# B&R Automation Studio project OpcUaSample410_BrbLibUa103 (part 5)

#### BrbDtStructCompare.c - Vergleicht zwei DtStructures
```c
/********************************************************************
 * COPYRIGHT -- Bernecker + Rainer
 ********************************************************************
 * Library: BrbLib
 * File: BrbDtStructCompare.c
 * Author: niedermeierr
 * Created: December 11, 2013
 ********************************************************************
 * Implementation of library BrbLib
 ********************************************************************/

#include <bur/plctypes.h>
#ifdef __cplusplus
	extern "C"
	{
#endif

	#include "BrbLib.h"

#ifdef __cplusplus
	};
#endif

// NOLINTBEGIN(readability-*, bugprone-easily-swappable-parameters, clang-diagnostic-invalid-utf8, clang-diagnostic-invalid-source-encoding, clang-diagnostic-pointer-arith, clang-diagnostic-strict-prototypes, hicpp-uppercase-literal-suffix, cppcoreguidelines-*, performance-*)

/* Vergleicht zwei DtStructures */
plcbit BrbDtStructCompare(struct DTStructure* pDtStruct1, enum BrbTimeAndDateCompare_ENUM eCompare, struct DTStructure* pDtStruct2) // NOLINT(readability-function-cognitive-complexity)
{
	// Prüfung der Parameter
	if(pDtStruct1 == 0)
	{
		return 0;
	}
	if(pDtStruct2 == 0)
	{
		return 0;
	}
	// Vergleich
	BOOL bResult = 0;
	switch(eCompare) // NOLINT(hicpp-multiway-paths-covered)
	{
		case eBRB_TAD_COMPARE_YOUNGER:
			if(pDtStruct1->year < pDtStruct2->year)
			{
				bResult = 1;
			}
			else if(pDtStruct1->year == pDtStruct2->year)
			{
				if(pDtStruct1->month < pDtStruct2->month)
				{
					bResult = 1;
				}
				else if(pDtStruct1->month == pDtStruct2->month)
				{
					if(pDtStruct1->day < pDtStruct2->day)
					{
						bResult = 1;
					}
					else if(pDtStruct1->day == pDtStruct2->day)
					{
						if(pDtStruct1->hour < pDtStruct2->hour)
						{
							bResult = 1;
						}
						else if(pDtStruct1->hour == pDtStruct2->hour)
						{
							if(pDtStruct1->minute < pDtStruct2->minute)
							{
								bResult = 1;
							}
							else if(pDtStruct1->minute == pDtStruct2->minute)
							{
								if(pDtStruct1->second < pDtStruct2->second)
								{
									bResult = 1;
								}
								else if(pDtStruct1->second == pDtStruct2->second)
								{
									if(pDtStruct1->millisec < pDtStruct2->millisec)
									{
										bResult = 1;
									}
									else if(pDtStruct1->millisec == pDtStruct2->millisec)
									{
										if(pDtStruct1->microsec < pDtStruct2->microsec)
										{
											bResult = 1;
										}
										else if(pDtStruct1->microsec == pDtStruct2->microsec)
										{
											bResult = 0;
										}
									}
								}
							}
						}
					}
				}
			}
			break;

		case eBRB_TAD_COMPARE_YOUNGEREQUAL:
			// NOLINTBEGIN(bugprone-branch-clone)
			if(pDtStruct1->year < pDtStruct2->year)
			{
				bResult = 1;
			}
			else if(pDtStruct1->year == pDtStruct2->year)
			{
				if(pDtStruct1->month < pDtStruct2->month)
				{
					bResult = 1;
				}
				else if(pDtStruct1->month == pDtStruct2->month)
				{
					if(pDtStruct1->day < pDtStruct2->day)
					{
						bResult = 1;
					}
					else if(pDtStruct1->day == pDtStruct2->day)
					{
						if(pDtStruct1->hour < pDtStruct2->hour)
						{
							bResult = 1;
						}
						else if(pDtStruct1->hour == pDtStruct2->hour)
						{
							if(pDtStruct1->minute < pDtStruct2->minute)
							{
								bResult = 1;
							}
							else if(pDtStruct1->minute == pDtStruct2->minute)
							{
								if(pDtStruct1->second < pDtStruct2->second)
								{
									bResult = 1;
								}
								else if(pDtStruct1->second == pDtStruct2->second)
								{
									if(pDtStruct1->millisec < pDtStruct2->millisec)
									{
										bResult = 1;
									}
									else if(pDtStruct1->millisec == pDtStruct2->millisec)
									{
										if(pDtStruct1->microsec < pDtStruct2->microsec)
										{
											bResult = 1;
										}
										else if(pDtStruct1->microsec == pDtStruct2->microsec)
										{
											bResult = 1;
										}
									}
								}
							}
						}
					}
				}
			}
			// NOLINTEND(bugprone-branch-clone)
			break;

		case eBRB_TAD_COMPARE_EQUAL:
			if((pDtStruct1->year == pDtStruct2->year) &&
				(pDtStruct1->month == pDtStruct2->month) &&
				(pDtStruct1->day == pDtStruct2->day) &&
				(pDtStruct1->hour == pDtStruct2->hour) &&
				(pDtStruct1->minute == pDtStruct2->minute) &&
				(pDtStruct1->second == pDtStruct2->second) &&
				(pDtStruct1->millisec == pDtStruct2->millisec) &&
				(pDtStruct1->microsec == pDtStruct2->microsec)
				)
			{
				bResult = 1;
			}
			break;

		case eBRB_TAD_COMPARE_OLDEREQUAL:
			// NOLINTBEGIN(bugprone-branch-clone)
			if(pDtStruct1->year > pDtStruct2->year)
			{
				bResult = 1;
			}
			else if(pDtStruct1->year == pDtStruct2->year)
			{
				if(pDtStruct1->month > pDtStruct2->month)
				{
					bResult = 1;
				}
				else if(pDtStruct1->month == pDtStruct2->month)
				{
					if(pDtStruct1->day > pDtStruct2->day)
					{
						bResult = 1;
					}
					else if(pDtStruct1->day == pDtStruct2->day)
					{
						if(pDtStruct1->hour > pDtStruct2->hour)
						{
							bResult = 1;
						}
						else if(pDtStruct1->hour == pDtStruct2->hour)
						{
							if(pDtStruct1->minute > pDtStruct2->minute)
							{
								bResult = 1;
							}
							else if(pDtStruct1->minute == pDtStruct2->minute)
							{
								if(pDtStruct1->second > pDtStruct2->second)
								{
									bResult = 1;
								}
								else if(pDtStruct1->second == pDtStruct2->second)
								{
									if(pDtStruct1->millisec > pDtStruct2->millisec)
									{
										bResult = 1;
									}
									else if(pDtStruct1->millisec == pDtStruct2->millisec)
									{
										if(pDtStruct1->microsec > pDtStruct2->microsec)
										{
											bResult = 1;
										}
										else if(pDtStruct1->microsec == pDtStruct2->microsec)
										{
											bResult = 1;
										}
									}
								}
							}
						}
					}
				}
			}
			// NOLINTEND(bugprone-branch-clone)
			break;

		case eBRB_TAD_COMPARE_OLDER:
			if(pDtStruct1->year > pDtStruct2->year)
			{
				bResult = 1;
			}
			else if(pDtStruct1->year == pDtStruct2->year)
			{
				if(pDtStruct1->month > pDtStruct2->month)
				{
					bResult = 1;
				}
				else if(pDtStruct1->month == pDtStruct2->month)
				{
					if(pDtStruct1->day > pDtStruct2->day)
					{
						bResult = 1;
					}
					else if(pDtStruct1->day == pDtStruct2->day)
					{
						if(pDtStruct1->hour > pDtStruct2->hour)
						{
							bResult = 1;
						}
						else if(pDtStruct1->hour == pDtStruct2->hour)
						{
							if(pDtStruct1->minute > pDtStruct2->minute)
							{
								bResult = 1;
							}
							else if(pDtStruct1->minute == pDtStruct2->minute)
							{
								if(pDtStruct1->second > pDtStruct2->second)
								{
									bResult = 1;
								}
								else if(pDtStruct1->second == pDtStruct2->second)
								{
									if(pDtStruct1->millisec > pDtStruct2->millisec)
									{
										bResult = 1;
									}
									else if(pDtStruct1->millisec == pDtStruct2->millisec)
									{
										if(pDtStruct1->microsec > pDtStruct2->microsec)
										{
											bResult = 1;
										}
										else if(pDtStruct1->microsec == pDtStruct2->microsec)
										{
											bResult = 0;
										}
									}
								}
							}
						}
					}
				}
			}
			break;

	}

	return bResult;
}

// NOLINTEND(readability-*, bugprone-easily-swappable-parameters, clang-diagnostic-invalid-utf8, clang-diagnostic-invalid-source-encoding, clang-diagnostic-pointer-arith, clang-diagnostic-strict-prototypes, hicpp-uppercase-literal-suffix, cppcoreguidelines-*, performance-*)
```

#### BrbDtStructAddDays.c - Addiert zu einer DTStructure die angegebenen Sekunden
```c
/********************************************************************
 * COPYRIGHT -- Bernecker + Rainer
 ********************************************************************
 * Library: BrbLib
 * File: BrbDtStructAddSeconds.c
 * Author: niedermeierr
 * Created: September 08, 2021
 ********************************************************************
 * Implementation of library BrbLib
 ********************************************************************/

#include <bur/plctypes.h>
#ifdef __cplusplus
	extern "C"
	{
#endif

#include "BrbLib.h"
#include <AnsiCFunc.h>

#ifdef __cplusplus
	};
#endif

// NOLINTBEGIN(readability-*, bugprone-easily-swappable-parameters, clang-diagnostic-invalid-utf8, clang-diagnostic-invalid-source-encoding, clang-diagnostic-pointer-arith, clang-diagnostic-strict-prototypes, hicpp-uppercase-literal-suffix, cppcoreguidelines-*, performance-*)

/* Addiert zu einer DTStructure die angegebenen Sekunden */
plcdt BrbDtStructAddDays(struct DTStructure* pDtStruct, signed long nDays)
{
	// Prüfung der Parameter
	if(pDtStruct == 0)
	{
		return 0;
	}
	// Addieren
	UINT nMilliSecondsBefore = pDtStruct->millisec;
	UINT nMicroSecondsBefore = pDtStruct->microsec;
	DATE_AND_TIME dtTime = DTStructure_TO_DT((UDINT)pDtStruct);
	// Es müssen Sekunden addiert werden. Durch eine Multiplikation der Stunden mit 60s*60m*24h = 86400s könnte der Bereich eines Dint nicht mehr ausreichen
	// Daher wird eine Schleife durchlaufen.
	UDINT nLoop = 0;
	if(nDays < 0)
	{
		for(nLoop=0; nLoop<(UDINT)abs(nDays); nLoop++)
		{
			dtTime = dtTime - nBRB_SECONDS_PER_DAY;
		}
	}
	else
	{
		for(nLoop=0; nLoop<(UDINT)abs(nDays); nLoop++)
		{
			dtTime = dtTime + nBRB_SECONDS_PER_DAY;
		}
	}
	DT_TO_DTStructure(dtTime, (UDINT)pDtStruct);
	pDtStruct->millisec = nMilliSecondsBefore;
	pDtStruct->microsec = nMicroSecondsBefore;
	return dtTime;
}

// NOLINTEND(readability-*, bugprone-easily-swappable-parameters, clang-diagnostic-invalid-utf8, clang-diagnostic-invalid-source-encoding, clang-diagnostic-pointer-arith, clang-diagnostic-strict-prototypes, hicpp-uppercase-literal-suffix, cppcoreguidelines-*, performance-*)
```

#### BrbDtStructAddHours.c - Addiert zu einer DTStructure die angegebenen Sekunden
```c
/********************************************************************
 * COPYRIGHT -- Bernecker + Rainer
 ********************************************************************
 * Library: BrbLib
 * File: BrbDtStructAddSeconds.c
 * Author: niedermeierr
 * Created: September 08, 2021
 ********************************************************************
 * Implementation of library BrbLib
 ********************************************************************/

#include <bur/plctypes.h>
#ifdef __cplusplus
	extern "C"
	{
#endif

#include "BrbLib.h"
#include <AnsiCFunc.h>

#ifdef __cplusplus
	};
#endif

// NOLINTBEGIN(readability-*, bugprone-easily-swappable-parameters, clang-diagnostic-invalid-utf8, clang-diagnostic-invalid-source-encoding, clang-diagnostic-pointer-arith, clang-diagnostic-strict-prototypes, hicpp-uppercase-literal-suffix, cppcoreguidelines-*, performance-*)

/* Addiert zu einer DTStructure die angegebenen Sekunden */
plcdt BrbDtStructAddHours(struct DTStructure* pDtStruct, signed long nHours)
{
	// Prüfung der Parameter
	if(pDtStruct == 0)
	{
		return 0;
	}
	// Addieren
	UINT nMilliSecondsBefore = pDtStruct->millisec;
	UINT nMicroSecondsBefore = pDtStruct->microsec;
	DATE_AND_TIME dtTime = DTStructure_TO_DT((UDINT)pDtStruct);
	// Es müssen Sekunden addiert werden. Durch eine Multiplikation der Stunden mit 60s*60m = 3600s könnte der Bereich eines Dint nicht mehr ausreichen
	// Daher wird eine Schleife durchlaufen.
	UDINT nLoop = 0;
	if(nHours < 0)
	{
		for(nLoop=0; nLoop<(UDINT)abs(nHours); nLoop++)
		{
			dtTime = dtTime - nBRB_SECONDS_PER_HOUR;
		}
	}
	else
	{
		for(nLoop=0; nLoop<(UDINT)abs(nHours); nLoop++)
		{
			dtTime = dtTime + nBRB_SECONDS_PER_HOUR;
		}
	}
	DT_TO_DTStructure(dtTime, (UDINT)pDtStruct);
	pDtStruct->millisec = nMilliSecondsBefore;
	pDtStruct->microsec = nMicroSecondsBefore;
	return dtTime;
}

// NOLINTEND(readability-*, bugprone-easily-swappable-parameters, clang-diagnostic-invalid-utf8, clang-diagnostic-invalid-source-encoding, clang-diagnostic-pointer-arith, clang-diagnostic-strict-prototypes, hicpp-uppercase-literal-suffix, cppcoreguidelines-*, performance-*)
```

#### BrbDtStructAddMinutes.c - Addiert zu einer DTStructure die angegebenen Sekunden
```c
/********************************************************************
 * COPYRIGHT -- Bernecker + Rainer
 ********************************************************************
 * Library: BrbLib
 * File: BrbDtStructAddSeconds.c
 * Author: niedermeierr
 * Created: September 08, 2021
 ********************************************************************
 * Implementation of library BrbLib
 ********************************************************************/

#include <bur/plctypes.h>
#ifdef __cplusplus
	extern "C"
	{
#endif

#include "BrbLib.h"
#include <AnsiCFunc.h>

#ifdef __cplusplus
	};
#endif

// NOLINTBEGIN(readability-*, bugprone-easily-swappable-parameters, clang-diagnostic-invalid-utf8, clang-diagnostic-invalid-source-encoding, clang-diagnostic-pointer-arith, clang-diagnostic-strict-prototypes, hicpp-uppercase-literal-suffix, cppcoreguidelines-*, performance-*)

/* Addiert zu einer DTStructure die angegebenen Sekunden */
plcdt BrbDtStructAddMinutes(struct DTStructure* pDtStruct, signed long nMinutes)
{
	// Prüfung der Parameter
	if(pDtStruct == 0)
	{
		return 0;
	}
	// Addieren
	UINT nMilliSecondsBefore = pDtStruct->millisec;
	UINT nMicroSecondsBefore = pDtStruct->microsec;
	DATE_AND_TIME dtTime = DTStructure_TO_DT((UDINT)pDtStruct);
	// Es müssen Sekunden addiert werden. Durch eine Multiplikation der Minuten mit 60s könnte der Bereich eines Dint nicht mehr ausreichen
	// Daher wird eine Schleife durchlaufen.
	UDINT nLoop = 0;
	if(nMinutes < 0)
	{
		for(nLoop=0; nLoop<(UDINT)abs(nMinutes); nLoop++)
		{
			dtTime = dtTime - nBRB_SECONDS_PER_MINUTE;
		}
	}
	else
	{
		for(nLoop=0; nLoop<(UDINT)abs(nMinutes); nLoop++)
		{
			dtTime = dtTime + nBRB_SECONDS_PER_MINUTE;
		}
	}
	DT_TO_DTStructure(dtTime, (UDINT)pDtStruct);
	pDtStruct->millisec = nMilliSecondsBefore;
	pDtStruct->microsec = nMicroSecondsBefore;
	return dtTime;
}

// NOLINTEND(readability-*, bugprone-easily-swappable-parameters, clang-diagnostic-invalid-utf8, clang-diagnostic-invalid-source-encoding, clang-diagnostic-pointer-arith, clang-diagnostic-strict-prototypes, hicpp-uppercase-literal-suffix, cppcoreguidelines-*, performance-*)
```

#### BrbDtStructAddSeconds.c - Addiert zu einer DTStructure die angegebenen Sekunden
```c
/********************************************************************
 * COPYRIGHT -- Bernecker + Rainer
 ********************************************************************
 * Library: BrbLib
 * File: BrbDtStructAddSeconds.c
 * Author: niedermeierr
 * Created: September 08, 2021
 ********************************************************************
 * Implementation of library BrbLib
 ********************************************************************/

#include <bur/plctypes.h>
#ifdef __cplusplus
	extern "C"
	{
#endif

	#include "BrbLib.h"

#ifdef __cplusplus
	};
#endif

// NOLINTBEGIN(readability-*, bugprone-easily-swappable-parameters, clang-diagnostic-invalid-utf8, clang-diagnostic-invalid-source-encoding, clang-diagnostic-pointer-arith, clang-diagnostic-strict-prototypes, hicpp-uppercase-literal-suffix, cppcoreguidelines-*, performance-*)

/* Addiert zu einer DTStructure die angegebenen Sekunden */
plcdt BrbDtStructAddSeconds(struct DTStructure* pDtStruct, signed long nSeconds)
{
	// Prüfung der Parameter
	if(pDtStruct == 0)
	{
		return 0;
	}
	// Addieren
	UINT nMilliSecondsBefore = pDtStruct->millisec;
	UINT nMicroSecondsBefore = pDtStruct->microsec;
	DATE_AND_TIME dtTime = DTStructure_TO_DT((UDINT)pDtStruct);
	if(nSeconds < 0)
	{
		dtTime = dtTime - (UDINT)(nSeconds * -1);
	}
	else
	{
		dtTime = dtTime + (UDINT)nSeconds;
	}
	DT_TO_DTStructure(dtTime, (UDINT)pDtStruct);
	pDtStruct->millisec = nMilliSecondsBefore;
	pDtStruct->microsec = nMicroSecondsBefore;
	return dtTime;
}

// NOLINTEND(readability-*, bugprone-easily-swappable-parameters, clang-diagnostic-invalid-utf8, clang-diagnostic-invalid-source-encoding, clang-diagnostic-pointer-arith, clang-diagnostic-strict-prototypes, hicpp-uppercase-literal-suffix, cppcoreguidelines-*, performance-*)
```

#### BrbDtStructAddMilliseconds.c - Addiert zu einer DTStructure die angegebenen Millisekunden
```c
/********************************************************************
 * COPYRIGHT -- Bernecker + Rainer
 ********************************************************************
 * Library: BrbLib
 * File: BrbDtStructAddMilliseconds.c
 * Author: niedermeierr
 * Created: December 11, 2013
 ********************************************************************
 * Implementation of library BrbLib
 ********************************************************************/

#include <bur/plctypes.h>
#ifdef __cplusplus
	extern "C"
	{
#endif

	#include "BrbLib.h"

#ifdef __cplusplus
	};
#endif

// NOLINTBEGIN(readability-*, bugprone-easily-swappable-parameters, clang-diagnostic-invalid-utf8, clang-diagnostic-invalid-source-encoding, clang-diagnostic-pointer-arith, clang-diagnostic-strict-prototypes, hicpp-uppercase-literal-suffix, cppcoreguidelines-*, performance-*)

/* Addiert zu einer DTStructure die angegebenen Millisekunden */
plcdt BrbDtStructAddMilliseconds(struct DTStructure* pDtStruct, signed long nMilliseconds)
{
	// Prüfung der Parameter
	if(pDtStruct == 0)
	{
		return 0;
	}
	// Addieren
	DINT nMilliSecondsBefore = (DINT)pDtStruct->millisec;
	UINT nMicroSecondsBefore = pDtStruct->microsec;
	DATE_AND_TIME dtTime = DTStructure_TO_DT((UDINT)pDtStruct);
	DINT nSeconds = (DINT)((REAL)nMilliseconds / (REAL)nBRB_MILLISECONDS_PER_SECOND);
	if(nSeconds < 0)
	{
		dtTime = dtTime - (UDINT)(nSeconds * -1);
	}
	else
	{
		dtTime = dtTime + (UDINT)nSeconds;
	}
	DINT nMillisecondsLeft = nMilliseconds - nSeconds * (DINT)nBRB_MILLISECONDS_PER_SECOND;
	if(nMilliSecondsBefore + nMillisecondsLeft >= (DINT)nBRB_MILLISECONDS_PER_SECOND)
	{
		dtTime += 1;
		nMillisecondsLeft -= (DINT)nBRB_MILLISECONDS_PER_SECOND;
	}
	else if(nMilliSecondsBefore + nMillisecondsLeft < 0)
	{
		dtTime -= 1;
		nMillisecondsLeft += (DINT)nBRB_MILLISECONDS_PER_SECOND;
	}
	DT_TO_DTStructure(dtTime, (UDINT)pDtStruct);
	pDtStruct->millisec = (UINT)(nMilliSecondsBefore + nMillisecondsLeft);
	pDtStruct->microsec = nMicroSecondsBefore;
	return dtTime;
}

// NOLINTEND(readability-*, bugprone-easily-swappable-parameters, clang-diagnostic-invalid-utf8, clang-diagnostic-invalid-source-encoding, clang-diagnostic-pointer-arith, clang-diagnostic-strict-prototypes, hicpp-uppercase-literal-suffix, cppcoreguidelines-*, performance-*)
```

#### BrbDtStructAddMillisecondsLReal.c - Addiert zu einer DTStructure die angegebenen Millisekunden
```c
/********************************************************************
 * COPYRIGHT -- Bernecker + Rainer
 ********************************************************************
 * Library: BrbLib
 * File: BrbDtStructAddMillisecondsLReal.c
 * Author: niedermeierr
 * Created: September 10, 2021
 ********************************************************************
 * Implementation of library BrbLib
 ********************************************************************/

#include <bur/plctypes.h>
#ifdef __cplusplus
	extern "C"
	{
#endif

	#include "BrbLib.h"

#ifdef __cplusplus
	};
#endif

// NOLINTBEGIN(readability-*, bugprone-easily-swappable-parameters, clang-diagnostic-invalid-utf8, clang-diagnostic-invalid-source-encoding, clang-diagnostic-pointer-arith, clang-diagnostic-strict-prototypes, hicpp-uppercase-literal-suffix, cppcoreguidelines-*, performance-*)

/* Addiert zu einer DTStructure die angegebenen Millisekunden */
plcdt BrbDtStructAddMillisecondsLReal(struct DTStructure* pDtStruct, double rMilliseconds)
{
	// Prüfung der Parameter
	if(pDtStruct == 0)
	{
		return 0;
	}
	// Addieren
	LREAL rDays = rMilliseconds / (LREAL)nBRB_MILLISECONDS_PER_DAY; // [ms/day]
	DINT nDays = (DINT)rDays; // Nachkomma-Stellen werden abgeschnitten
	BrbDtStructAddDays(pDtStruct, nDays);
	rMilliseconds -= (LREAL)nDays * (LREAL)nBRB_MILLISECONDS_PER_DAY;
	DINT nMilliseconds = (DINT)rMilliseconds;
	BrbDtStructAddMilliseconds(pDtStruct, nMilliseconds);
	DATE_AND_TIME dtTime = DTStructure_TO_DT((UDINT)pDtStruct);
	return dtTime;
}

// NOLINTEND(readability-*, bugprone-easily-swappable-parameters, clang-diagnostic-invalid-utf8, clang-diagnostic-invalid-source-encoding, clang-diagnostic-pointer-arith, clang-diagnostic-strict-prototypes, hicpp-uppercase-literal-suffix, cppcoreguidelines-*, performance-*)
```

#### BrbGetTimeTextMs.c - Gibt die angebenene Millisekunden-Zeit alsText zurück
```c
/********************************************************************
 * COPYRIGHT -- Bernecker + Rainer
 ********************************************************************
 * Library: BrbLib
 * File: BrbGetTimeTextMs.c
 * Author: niedermeierr
 * Created: April 29, 2016
 ********************************************************************
 * Implementation of library BrbLib
 ********************************************************************/

#include <bur/plctypes.h>
#ifdef __cplusplus
	extern "C"
	{
#endif

#include "BrbLib.h"
#include <string.h>

#ifdef __cplusplus
	};
#endif

// NOLINTBEGIN(readability-*, bugprone-easily-swappable-parameters, clang-diagnostic-invalid-utf8, clang-diagnostic-invalid-source-encoding, clang-diagnostic-pointer-arith, clang-diagnostic-strict-prototypes, hicpp-uppercase-literal-suffix, cppcoreguidelines-*, performance-*)

/* Gibt die angebenene Millisekunden-Zeit als Text zurück */
unsigned short BrbGetTimeTextMs(signed long nMilliseconds, plcstring* pText, unsigned long nTextSize, plcstring* pFormat, plcbit bClip) // NOLINT(readability-function-cognitive-complexity)
{
	// Prüfung der Parameter
	if(pText == 0)
	{
		return eBRB_ERR_NULL_POINTER;
	}
	if(nTextSize == 0)
	{
		return eBRB_ERR_INVALID_PARAMETER;
	}
	if(pFormat == 0)
	{
		return eBRB_ERR_NULL_POINTER;
	}
	// Text ermitteln
	BrbStringCopy(pText, pFormat, nTextSize);
	STRING sItoA[20];
	memset((USINT*)sItoA, 0, sizeof(sItoA));
	if(BrbStringGetAdrOf(pText, "dd", 0) != 0)
	{
		DINT nDays = nMilliseconds / (DINT)nBRB_MILLISECONDS_PER_DAY;
		nMilliseconds -= nDays * (DINT)nBRB_MILLISECONDS_PER_DAY;
		brsitoa(nDays, (UDINT)&sItoA);
		if(nDays < 10)
		{
			BrbStringInsert(sItoA, 0, "0");
		}
		BrbStringReplace(pText, "dd", sItoA);
	}
	else if(BrbStringGetAdrOf(pText, "d", 0) != 0)
	{
		DINT nDays = nMilliseconds / (DINT)nBRB_MILLISECONDS_PER_DAY;
		nMilliseconds -= nDays * (DINT)nBRB_MILLISECONDS_PER_DAY;
		brsitoa(nDays, (UDINT)&sItoA);
		BrbStringReplace(pText, "d", sItoA);
	}
	else if(bClip == 1)
	{
		DINT nDays = nMilliseconds / (DINT)nBRB_MILLISECONDS_PER_DAY;
		nMilliseconds -= nDays * (DINT)nBRB_MILLISECONDS_PER_DAY;
	}
	if(BrbStringGetAdrOf(pText, "hh", 0) != 0)
	{
		DINT nHours = nMilliseconds / (DINT)nBRB_MILLISECONDS_PER_HOUR;
		nMilliseconds -= nHours * (DINT)nBRB_MILLISECONDS_PER_HOUR;
		brsitoa(nHours, (UDINT)&sItoA);
		if(nHours < 10)
		{
			BrbStringInsert(sItoA, 0, "0");
		}
		BrbStringReplace(pText, "hh", sItoA);
	}
	else if(BrbStringGetAdrOf(pText, "h", 0) != 0)
	{
		DINT nHours = nMilliseconds / (DINT)nBRB_MILLISECONDS_PER_HOUR;
		nMilliseconds -= nHours * (DINT)nBRB_MILLISECONDS_PER_HOUR;
		brsitoa(nHours, (UDINT)&sItoA);
		BrbStringReplace(pText, "h", sItoA);
	}
	else if(bClip == 1)
	{
		DINT nHours = nMilliseconds / (DINT)nBRB_MILLISECONDS_PER_HOUR;
		nMilliseconds -= nHours * (DINT)nBRB_MILLISECONDS_PER_HOUR;
	}
	if(BrbStringGetAdrOf(pText, "MM", 0) != 0)
	{
		DINT nMinutes = nMilliseconds / (DINT)nBRB_MILLISECONDS_PER_MINUTE;
		nMilliseconds -= nMinutes * (DINT)nBRB_MILLISECONDS_PER_MINUTE;
		brsitoa(nMinutes, (UDINT)&sItoA);
		if(nMinutes < 10)
		{
			BrbStringInsert(sItoA, 0, "0");
		}
		BrbStringReplace(pText, "MM", sItoA);
	}
	else if(BrbStringGetAdrOf(pText, "M", 0) != 0)
	{
		DINT nMinutes = nMilliseconds / (DINT)nBRB_MILLISECONDS_PER_MINUTE;
		nMilliseconds -= nMinutes * (DINT)nBRB_MILLISECONDS_PER_MINUTE;
		brsitoa(nMinutes, (UDINT)&sItoA);
		BrbStringReplace(pText, "M", sItoA);
	}
	else if(bClip == 1)
	{
		DINT nMinutes = nMilliseconds / (DINT)nBRB_MILLISECONDS_PER_MINUTE;
		nMilliseconds -= nMinutes * (DINT)nBRB_MILLISECONDS_PER_MINUTE;
	}
	if(BrbStringGetAdrOf(pText, "ss", 0) != 0)
	{
		DINT nSeconds = nMilliseconds / (DINT)nBRB_MILLISECONDS_PER_SECOND;
		nMilliseconds -= nSeconds * (DINT)nBRB_MILLISECONDS_PER_SECOND;
		brsitoa(nSeconds, (UDINT)&sItoA);
		if(nSeconds < 10)
		{
			BrbStringInsert(sItoA, 0, "0");
		}
		BrbStringReplace(pText, "ss", sItoA);
	}
	else if(BrbStringGetAdrOf(pText, "s", 0) != 0)
	{
		DINT nSeconds = nMilliseconds / (DINT)nBRB_MILLISECONDS_PER_SECOND;
		nMilliseconds -= nSeconds * (DINT)nBRB_MILLISECONDS_PER_SECOND;
		brsitoa((DINT)nSeconds, (UDINT)&sItoA);
		BrbStringReplace(pText, "s", sItoA);
	}
	else if(bClip == 1)
	{
		DINT nSeconds = nMilliseconds / (DINT)nBRB_MILLISECONDS_PER_SECOND;
		nMilliseconds -= nSeconds * (DINT)nBRB_MILLISECONDS_PER_SECOND;
	}
	if(BrbStringGetAdrOf(pText, "mil", 0) != 0)
	{
		brsitoa(nMilliseconds, (UDINT)&sItoA);
		if(nMilliseconds < 10)
		{
			BrbStringInsert(sItoA, 0, "00");
		}
		else if(nMilliseconds < 100)
		{
			BrbStringInsert(sItoA, 0, "0");
		}
		BrbStringReplace(pText, "mil", sItoA);
	}
	return eBRB_ERR_OK;
}

// NOLINTEND(readability-*, bugprone-easily-swappable-parameters, clang-diagnostic-invalid-utf8, clang-diagnostic-invalid-source-encoding, clang-diagnostic-pointer-arith, clang-diagnostic-strict-prototypes, hicpp-uppercase-literal-suffix, cppcoreguidelines-*, performance-*)
```

#### BrbGetTimeDiffMsDtStruct.c - Gibt die Zeit-Differenz zweier DTStruct-Zeiten in [ms] zurück
```c
/********************************************************************
 * COPYRIGHT -- Bernecker + Rainer
 ********************************************************************
 * Library: BrbLib
 * File: BrbGetTimeDiffMsDtStruct.c
 * Author: niedermeierr
 * Created: February 13, 2017
 ********************************************************************
 * Implementation of library BrbLib
 ********************************************************************/

#include <bur/plctypes.h>
#ifdef __cplusplus
	extern "C"
	{
#endif

#include "BrbLib.h"

#ifdef __cplusplus
	};
#endif

// NOLINTBEGIN(readability-*, bugprone-easily-swappable-parameters, clang-diagnostic-invalid-utf8, clang-diagnostic-invalid-source-encoding, clang-diagnostic-pointer-arith, clang-diagnostic-strict-prototypes, hicpp-uppercase-literal-suffix, cppcoreguidelines-*, performance-*)

/* Gibt die Zeit-Differenz zweier DtStruct-Zeiten in [ms] zurück */
signed long BrbGetTimeDiffMsDtStruct(struct DTStructure* pTimeStampBase, struct DTStructure* pTimeStampCompare)
{
	// Prüfung der Parameter
	if(pTimeStampBase == 0)
	{
		return 0;
	}
	if(pTimeStampCompare == 0)
	{
		return 0;
	}
	// Diff
	DINT nDiffMs = 0;
	DATE_AND_TIME dtTimeBase = DTStructure_TO_DT((UDINT)pTimeStampBase);
	DATE_AND_TIME dtTimeCompare = DTStructure_TO_DT((UDINT)pTimeStampCompare);
	UDINT nDiffS = 0;
	if(dtTimeBase >= dtTimeCompare)
	{
		nDiffS = DiffDT(dtTimeBase, dtTimeCompare);
		nDiffMs = (DINT)(pTimeStampCompare->millisec - pTimeStampBase->millisec);
		nDiffMs += (DINT)nDiffS * -(DINT)nBRB_MILLISECONDS_PER_SECOND;
	}
	else
	{
		nDiffS = DiffDT(dtTimeCompare, dtTimeBase);
		nDiffMs = (DINT)(pTimeStampCompare->millisec - pTimeStampBase->millisec);
		nDiffMs += (DINT)nDiffS * (DINT)nBRB_MILLISECONDS_PER_SECOND;
	}
	return nDiffMs;
}

// NOLINTEND(readability-*, bugprone-easily-swappable-parameters, clang-diagnostic-invalid-utf8, clang-diagnostic-invalid-source-encoding, clang-diagnostic-pointer-arith, clang-diagnostic-strict-prototypes, hicpp-uppercase-literal-suffix, cppcoreguidelines-*, performance-*)
```

#### BrbGetWeekdayDtStruct.c - Ermittelt den Wochentag einer DTStructure
```c
/********************************************************************
 * COPYRIGHT -- Bernecker + Rainer
 ********************************************************************
 * Library: BrbLib
 * File: BrbGetWeekdayDt.c
 * Author: niedermeierr
 * Created: May 17, 2021
 ********************************************************************
 * Implementation of library BrbLib
 ********************************************************************/

#include <bur/plctypes.h>
#ifdef __cplusplus
	extern "C"
	{
#endif

#include "BrbLib.h"

#ifdef __cplusplus
	};
#endif

// NOLINTBEGIN(readability-*, bugprone-easily-swappable-parameters, clang-diagnostic-invalid-utf8, clang-diagnostic-invalid-source-encoding, clang-diagnostic-pointer-arith, clang-diagnostic-strict-prototypes, hicpp-uppercase-literal-suffix, cppcoreguidelines-*, performance-*)

/* Ermittelt den Wochentag einer DTStructure */
BrbWeekdays_ENUM BrbGetWeekdayDtStruct(struct DTStructure* pDtStruct)
{
	UINT nMilliSecondsBefore = pDtStruct->millisec;
	UINT nMicroSecondsBefore = pDtStruct->microsec;
	DATE_AND_TIME dtTime = DTStructure_TO_DT((UDINT)pDtStruct);
	DT_TO_DTStructure(dtTime, (UDINT)pDtStruct);
	pDtStruct->millisec = nMilliSecondsBefore;
	pDtStruct->microsec = nMicroSecondsBefore;
	return (BrbWeekdays_ENUM)pDtStruct->wday;
}

// NOLINTEND(readability-*, bugprone-easily-swappable-parameters, clang-diagnostic-invalid-utf8, clang-diagnostic-invalid-source-encoding, clang-diagnostic-pointer-arith, clang-diagnostic-strict-prototypes, hicpp-uppercase-literal-suffix, cppcoreguidelines-*, performance-*)
```

#### BrbGetWeekdayDt.c - Ermittelt den Wochentag einer DATE_AND_TIME
```c
/********************************************************************
 * COPYRIGHT -- Bernecker + Rainer
 ********************************************************************
 * Library: BrbLib
 * File: BrbGetWeekdayDt.c
 * Author: niedermeierr
 * Created: May 17, 2021
 ********************************************************************
 * Implementation of library BrbLib
 ********************************************************************/

#include <bur/plctypes.h>
#ifdef __cplusplus
	extern "C"
	{
#endif

#include "BrbLib.h"

#ifdef __cplusplus
	};
#endif

// NOLINTBEGIN(readability-*, bugprone-easily-swappable-parameters, clang-diagnostic-invalid-utf8, clang-diagnostic-invalid-source-encoding, clang-diagnostic-pointer-arith, clang-diagnostic-strict-prototypes, hicpp-uppercase-literal-suffix, cppcoreguidelines-*, performance-*)

/* Gibt den Wochentag einer DT-Zeit zurück */
BrbWeekdays_ENUM BrbGetWeekdayDt(plcdt dtTime)
{
	DTStructure DtStruct;
	DT_TO_DTStructure(dtTime, (UDINT)&DtStruct);
	return (BrbWeekdays_ENUM)DtStruct.wday;
}

// NOLINTEND(readability-*, bugprone-easily-swappable-parameters, clang-diagnostic-invalid-utf8, clang-diagnostic-invalid-source-encoding, clang-diagnostic-pointer-arith, clang-diagnostic-strict-prototypes, hicpp-uppercase-literal-suffix, cppcoreguidelines-*, performance-*)
```

#### BrbTimerSwitch.c - Zeitschaltuhr für einen Kanal
```c
/********************************************************************
 * COPYRIGHT -- Bernecker + Rainer
 ********************************************************************
 * Library: BrbLib
 * File: BrbTimerSwitch.c
 * Author: niedermeierr
 * Created: January 22, 2016
 ********************************************************************
 * Implementation of library BrbLib
 ********************************************************************/

#include <bur/plctypes.h>
#ifdef __cplusplus
	extern "C"
	{
#endif

#include "BrbLib.h"
#include <string.h>

#ifdef __cplusplus
	};
#endif

// NOLINTBEGIN(readability-*, bugprone-easily-swappable-parameters, clang-diagnostic-invalid-utf8, clang-diagnostic-invalid-source-encoding, clang-diagnostic-pointer-arith, clang-diagnostic-strict-prototypes, hicpp-uppercase-literal-suffix, cppcoreguidelines-*, performance-*)

void SwitchOutputByType(struct BrbTimerSwitch* inst, BrbTimerSwitchType_ENUM eSwitchType);

/* Zeitschaltuhr für einen Kanal */
void BrbTimerSwitch(struct BrbTimerSwitch* inst) // NOLINT(readability-function-cognitive-complexity)
{
	// Zeitschaltuhr
	if(inst->bEnable == 1)
	{
		if(inst->pUserTime == 0)
		{
			inst->fbDTStructureGetTime.enable = 1;
			inst->fbDTStructureGetTime.pDTStructure = (UDINT)&inst->dtsUsedTime;
			DTStructureGetTime(&inst->fbDTStructureGetTime);
		}
		else
		{
			memcpy(&inst->dtsUsedTime, inst->pUserTime, sizeof(DTStructure));
		}
		if(inst->bClearOutOnNextCycle == 1)
		{
			inst->bClearOutOnNextCycle = 0;
			inst->bOut = 0;
		}
		if(inst->bCmdSwitchOff == 1)
		{
			inst->bCmdSwitchOff = 0;
			inst->bOut = 0;
		}
		else if(inst->bCmdSwitchOn == 1)
		{
			inst->bCmdSwitchOn = 0;
			inst->bOut = 1;
		}
		else if(inst->bCmdToggle == 1)
		{
			inst->bCmdToggle = 0;
			inst->bOut = !inst->bOut;
		}
		UINT nTimePointIndex = 0;
		for(nTimePointIndex=0; nTimePointIndex<=nBRB_TIMERSWITCH_POINT_INDEX_MAX; nTimePointIndex++)
		{
			BrbTimerSwitchParTimePoint_TYP* pTimePoint = &inst->Parameter.TimePoint[nTimePointIndex];
			if(pTimePoint->bActive == 1)
			{
				switch(inst->Parameter.eMode)
				{
					case eBRB_TIMERSWITCH_MODE_MONTH:
						if(inst->dtsUsedTime.month == pTimePoint->dtsTimePoint.month && inst->dtsUsedTime.day == pTimePoint->dtsTimePoint.day && inst->dtsUsedTime.hour == pTimePoint->dtsTimePoint.hour && inst->dtsUsedTime.minute == pTimePoint->dtsTimePoint.minute && inst->dtsUsedTime.second == pTimePoint->dtsTimePoint.second)
						{
							if(inst->bLocked == 0)
							{
								SwitchOutputByType(inst, pTimePoint->eSwitchType);
								inst->bLocked = 1; // Nach diesem Schalten müssen andere Schaltungen für 1 Sekunde gesperrt werden
							}
						}
						break;

					case eBRB_TIMERSWITCH_MODE_WEEK:
						if(inst->dtsUsedTime.wday == pTimePoint->dtsTimePoint.wday && inst->dtsUsedTime.hour == pTimePoint->dtsTimePoint.hour && inst->dtsUsedTime.minute == pTimePoint->dtsTimePoint.minute && inst->dtsUsedTime.second == pTimePoint->dtsTimePoint.second)
						{
							if(inst->bLocked == 0)
							{
								SwitchOutputByType(inst, pTimePoint->eSwitchType);
								inst->bLocked = 1; // Nach diesem Schalten müssen andere Schaltungen für 1 Sekunde gesperrt werden
							}
						}
						break;

					case eBRB_TIMERSWITCH_MODE_DAY:
						if(inst->dtsUsedTime.day == pTimePoint->dtsTimePoint.day && inst->dtsUsedTime.hour == pTimePoint->dtsTimePoint.hour && inst->dtsUsedTime.minute == pTimePoint->dtsTimePoint.minute && inst->dtsUsedTime.second == pTimePoint->dtsTimePoint.second)
						{
							if(inst->bLocked == 0)
							{
								SwitchOutputByType(inst, pTimePoint->eSwitchType);
								inst->bLocked = 1; // Nach diesem Schalten müssen andere Schaltungen für 1 Sekunde gesperrt werden
							}
						}
						break;

					case eBRB_TIMERSWITCH_MODE_HOUR:
						if(inst->dtsUsedTime.hour == pTimePoint->dtsTimePoint.hour && inst->dtsUsedTime.minute == pTimePoint->dtsTimePoint.minute && inst->dtsUsedTime.second == pTimePoint->dtsTimePoint.second)
						{
							if(inst->bLocked == 0)
							{
								SwitchOutputByType(inst, pTimePoint->eSwitchType);
								inst->bLocked = 1; // Nach diesem Schalten müssen andere Schaltungen für 1 Sekunde gesperrt werden
							}
						}
						break;

					case eBRB_TIMERSWITCH_MODE_MINUTE:
						if(inst->dtsUsedTime.minute == pTimePoint->dtsTimePoint.minute && inst->dtsUsedTime.second == pTimePoint->dtsTimePoint.second)
						{
							if(inst->bLocked == 0)
							{
								SwitchOutputByType(inst, pTimePoint->eSwitchType);
								inst->bLocked = 1; // Nach diesem Schalten müssen andere Schaltungen für 1 Sekunde gesperrt werden
							}
						}
						break;

					case eBRB_TIMERSWITCH_MODE_SECOND:
						if(inst->dtsUsedTime.second == pTimePoint->dtsTimePoint.second)
						{
							if(inst->bLocked == 0)
							{
								SwitchOutputByType(inst, pTimePoint->eSwitchType);
								inst->bLocked = 1; // Nach diesem Schalten müssen andere Schaltungen für 1 Sekunde gesperrt werden
							}
						}
						break;
				}
			}
		}
		inst->fbLock.IN = inst->bLocked;
		inst->fbLock.PT = 1000; // = 1s
		TON(&inst->fbLock);
		if(inst->fbLock.Q == 1)
		{
			inst->fbLock.IN = 0;
			inst->bLocked = 0;
		}
	}
}

void SwitchOutputByType(struct BrbTimerSwitch* inst, BrbTimerSwitchType_ENUM eSwitchType)
{
	switch(eSwitchType) // NOLINT(hicpp-multiway-paths-covered)
	{
		case eBRB_TIMERSWITCH_TYPE_OFF:
			inst->bOut = 0;
			inst->nSwitchCount += 1;
			break;

		case eBRB_TIMERSWITCH_TYPE_ON:
			inst->bOut = 1;
			inst->nSwitchCount += 1;
			break;

		case eBRB_TIMERSWITCH_TYPE_TOGGLE:
			inst->bOut = !inst->bOut;
			inst->nSwitchCount += 1;
			break;

		case eBRB_TIMERSWITCH_TYPE_IMPULSE:
			inst->bOut = 1;
			inst->nSwitchCount += 1;
			inst->bClearOutOnNextCycle = 1;
			break;

	}
}

// NOLINTEND(readability-*, bugprone-easily-swappable-parameters, clang-diagnostic-invalid-utf8, clang-diagnostic-invalid-source-encoding, clang-diagnostic-pointer-arith, clang-diagnostic-strict-prototypes, hicpp-uppercase-literal-suffix, cppcoreguidelines-*, performance-*)
```

#### Package Logical/Libraries/BrbLib/Strings - String-Funktionen

#### BrbUsintToHex.c - Wandelt einen Udint in einen Hex-String
```c
/********************************************************************
 * COPYRIGHT -- Bernecker + Rainer
 ********************************************************************
 * Library: BrbLib
 * File: BrbUdintToHex.c
 * Author: niedermeierr
 * Created: July 14, 2021
 ********************************************************************
 * Implementation of library BrbLib
 ********************************************************************/

#include <bur/plctypes.h>
#ifdef __cplusplus
	extern "C"
	{
#endif

#include "BrbLib.h"
#include <math.h>
#include <string.h>

#ifdef __cplusplus
	};
#endif

// NOLINTBEGIN(readability-*, bugprone-easily-swappable-parameters, clang-diagnostic-invalid-utf8, clang-diagnostic-invalid-source-encoding, clang-diagnostic-pointer-arith, clang-diagnostic-strict-prototypes, hicpp-uppercase-literal-suffix, cppcoreguidelines-*, performance-*)

/* Wandelt einen Usint in einen Hex-String */
unsigned short BrbUsintToHex(unsigned char nValue, plcstring* pHex, unsigned long nHexSize, plcbit bWithPraefix)
{
	memset(pHex, 0, nHexSize);
	if(bWithPraefix == 1)
	{
		BrbStringCat(pHex, "0x", nHexSize);
	}
	DINT nDigit = 0;
	for(nDigit=1; nDigit>=0; nDigit--)
	{
		UDINT nHelp1 = (UDINT)0xF << (UDINT)nDigit * 4; // NOLINT(hicpp-signed-bitwise)
		UDINT nHelp2 = nValue & nHelp1;
		UDINT nHelp3 = nHelp2 >> (UDINT)nDigit * 4;

		if(nHelp3 <= 9)
		{
			STRING sChar[2];
			sChar[0] = (char)(48 + nHelp3);
			sChar[1] = 0;
			BrbStringCat(pHex, sChar, nHexSize);
		}
		else
		{
			STRING sChar[2];
			sChar[0] = (char)(65 + nHelp3 - 10);
			sChar[1] = 0;
			BrbStringCat(pHex, sChar, nHexSize);
		}
	}
	return eBRB_ERR_OK;
}

// NOLINTEND(readability-*, bugprone-easily-swappable-parameters, clang-diagnostic-invalid-utf8, clang-diagnostic-invalid-source-encoding, clang-diagnostic-pointer-arith, clang-diagnostic-strict-prototypes, hicpp-uppercase-literal-suffix, cppcoreguidelines-*, performance-*)
```

#### BrbUsintArrayToHex.c
```c
/********************************************************************
 * COPYRIGHT -- Bernecker + Rainer
 ********************************************************************
 * Library: BrbLib
 * File: BrbUdintToHex.c
 * Author: niedermeierr
 * Created: July 14, 2021
 ********************************************************************
 * Implementation of library BrbLib
 ********************************************************************/

#include <bur/plctypes.h>
#ifdef __cplusplus
	extern "C"
	{
#endif

#include "BrbLib.h"
#include <string.h>

#ifdef __cplusplus
	};
#endif

// NOLINTBEGIN(readability-*, bugprone-easily-swappable-parameters, clang-diagnostic-invalid-utf8, clang-diagnostic-invalid-source-encoding, clang-diagnostic-pointer-arith, clang-diagnostic-strict-prototypes, hicpp-uppercase-literal-suffix, cppcoreguidelines-*, performance-*)

/* Wandelt ein Usint-Array in einen Hex-String */
unsigned short BrbUsintArrayToHex(unsigned char* pArray, signed long nArrayLength, plcstring* pHex, unsigned long nHexSize, plcbit bDescending)
{
	UINT nStatus = eBRB_ERR_OK;
	if(pHex != 0)
	{
		memset(pHex, 0, nHexSize);
		UDINT nTextOffset = 0;
		if(nArrayLength > 0)
		{
			if(bDescending == 0)
			{
				// Aufsteigend
				UDINT nIndex = 0;
				for(nIndex=0; nIndex<(UDINT)nArrayLength; nIndex++)
				{
					USINT nValue = *(pArray+nIndex);
					STRING sValueHexUsint[16];
					BrbUsintToHex(nValue, sValueHexUsint, sizeof(sValueHexUsint), 0);
					BrbStringAppend(pHex, sValueHexUsint, &nTextOffset);
				}
			}
			else
			{
				// Absteigend
				DINT nIndex = 0;
				for(nIndex=(DINT)nArrayLength-1; nIndex>-1; nIndex--)
				{
					USINT nValue = *(pArray+nIndex);
					STRING sValueHexUsint[16];
					BrbUsintToHex(nValue, sValueHexUsint, sizeof(sValueHexUsint), 0);
					BrbStringAppend(pHex, sValueHexUsint, &nTextOffset);
				}
			}
		}
		else
		{
			nStatus = eBRB_ERR_INVALID_PARAMETER;
		}
	}
	else
	{
		nStatus = eBRB_ERR_NULL_POINTER;
	}
	return nStatus;
}

// NOLINTEND(readability-*, bugprone-easily-swappable-parameters, clang-diagnostic-invalid-utf8, clang-diagnostic-invalid-source-encoding, clang-diagnostic-pointer-arith, clang-diagnostic-strict-prototypes, hicpp-uppercase-literal-suffix, cppcoreguidelines-*, performance-*)
```

#### BrbHexToUsintArray.c - Wandelt ein Byte-Array in einen Hex-String
```c
/********************************************************************
 * COPYRIGHT -- Bernecker + Rainer
 ********************************************************************
 * Library: BrbLib
 * File: BrbUdintToHex.c
 * Author: niedermeierr
 * Created: July 14, 2021
 ********************************************************************
 * Implementation of library BrbLib
 ********************************************************************/

#include <bur/plctypes.h>
#ifdef __cplusplus
	extern "C"
	{
#endif

#include "BrbLib.h"
#include <string.h>

#ifdef __cplusplus
	};
#endif

// NOLINTBEGIN(readability-*, bugprone-easily-swappable-parameters, clang-diagnostic-invalid-utf8, clang-diagnostic-invalid-source-encoding, clang-diagnostic-pointer-arith, clang-diagnostic-strict-prototypes, hicpp-uppercase-literal-suffix, cppcoreguidelines-*, performance-*)

/* Wandelt einen Hex-String in ein Usint-Array */
unsigned short BrbHexToUsintArray(plcstring* pHex, unsigned char* pArray, signed long nArrayLength, plcbit bDescending) // NOLINT(readability-function-cognitive-complexity)
{
	UINT nStatus = eBRB_ERR_OK;
	if(pHex != 0 && pArray != 0)
	{
		if(nArrayLength > 0)
		{
			memset(pArray, 0, (UDINT)nArrayLength);
			UDINT nLengthHex = brsstrlen((UDINT)pHex);
			if(bDescending == 0)
			{
				BOOL bExpandFirstHex = 0;
				if(nLengthHex % 2 != 0)
				{
					// Ungerade Anzahl von Hex-Zeichen -> dem ersten Hex-Wert eine 0 voranstellen
					bExpandFirstHex = 1;
				}
				BOOL bLeave = 0;
				UDINT nCharIndex = 0;
				DINT nByteIndex = 0;
				STRING sValueHexUsint[4];
				UDINT nValueUdint = 0;
				do
				{
					if(nCharIndex >= nLengthHex || nByteIndex >= nArrayLength)
					{
						bLeave = 1;
					}
					else
					{
						// Das erste Byte könnte aus nur einem Hex-Zeichen bestehen
						if(nCharIndex == 0 && bExpandFirstHex == 1)
						{
							// Dem ersten Hex-Wert eine 0 voranstellen
							BrbStringGetSubText(pHex, nCharIndex, 1, sValueHexUsint);
							BrbStringInsert(sValueHexUsint, 0, "0");
							nValueUdint = BrbHexToUdint(sValueHexUsint);
							*(pArray + nByteIndex) = (USINT)nValueUdint;
							nCharIndex += 1;
						}
						else
						{
							BrbStringGetSubText(pHex, nCharIndex, 2, sValueHexUsint);
							nValueUdint = BrbHexToUdint(sValueHexUsint);
							*(pArray + nByteIndex) = (USINT)nValueUdint;
							nCharIndex += 2;
						}
						nByteIndex += 1;
					}
				} while(bLeave == 0);
			}
			else
			{
				BOOL bLeave = 0;
				DINT nCharIndex = (DINT)nLengthHex - 2;
				DINT nByteIndex = 0;
				STRING sValueHexUsint[4];
				UDINT nValueUdint = 0;
				do
				{
					if(nCharIndex < -1 || nByteIndex >= nArrayLength)
					{
						bLeave = 1;
					}
					else if(nCharIndex == -1)
					{
						// Das letzte Byte könnte aus nur einem Hex-Zeichen bestehen
						nCharIndex = 0;
						BrbStringGetSubText(pHex, (UDINT)nCharIndex, 1, sValueHexUsint);
						BrbStringInsert(sValueHexUsint, 0, "0");
						nValueUdint = BrbHexToUdint(sValueHexUsint);
						*(pArray + nByteIndex) = (USINT)nValueUdint;
						bLeave = 1;
					}
					else
					{
						BrbStringGetSubText(pHex, (UDINT)nCharIndex, 2, sValueHexUsint);
						nValueUdint = BrbHexToUdint(sValueHexUsint);
						*(pArray + nByteIndex) = (USINT)nValueUdint;
						nCharIndex -= 2;
						nByteIndex += 1;
					}
				} while(bLeave == 0);
			}
		}
		else
		{
			nStatus = eBRB_ERR_INVALID_PARAMETER;
		}
	}
	else
	{
		nStatus = eBRB_ERR_NULL_POINTER;
	}
	return nStatus;
}

// NOLINTEND(readability-*, bugprone-easily-swappable-parameters, clang-diagnostic-invalid-utf8, clang-diagnostic-invalid-source-encoding, clang-diagnostic-pointer-arith, clang-diagnostic-strict-prototypes, hicpp-uppercase-literal-suffix, cppcoreguidelines-*, performance-*)
```

#### BrbUdintToAscii.c - Wandelt einen UDINT-Wert zu einem String
```c
/********************************************************************
 * COPYRIGHT -- Bernecker + Rainer
 ********************************************************************
 * Library: BrbLib
 * File: BrbUdintToAscii.c
 * Author: niedermeierr
 * Created: June 11, 2013
 ********************************************************************
 * Implementation of library BrbLib
 ********************************************************************/

#include <bur/plctypes.h>
#ifdef __cplusplus
	extern "C"
	{
#endif

#include "BrbLib.h"

#ifdef __cplusplus
	};
#endif

// NOLINTBEGIN(readability-*, bugprone-easily-swappable-parameters, clang-diagnostic-invalid-utf8, clang-diagnostic-invalid-source-encoding, clang-diagnostic-pointer-arith, clang-diagnostic-strict-prototypes, hicpp-uppercase-literal-suffix, cppcoreguidelines-*, performance-*)

/* Wandelt einen UDINT-Wert zu einem String */
unsigned short BrbUdintToAscii(unsigned long nValue, plcstring* pText)
{
	UDINT nDiff = 0; // Wertigkeit
	UDINT nHelpVal = 0;
	BOOL bFirstDigitFound = 0; // Erste gültige Stelle erkannt
	// Die Schleife beginnt mit der größten Stelle und geht runter bis zur zweitletzten Stelle (Wertigkeit 10-90)
	for(nDiff = 1000000000; nDiff > 1; )
	{
		nHelpVal = nValue/nDiff;		// Ganzzahldivision bringt die Wertigkeit der gewünschten Stelle
		// Führende Nullen werden unterdrückt
		if(nHelpVal > 0 || bFirstDigitFound == 1)
		{
			bFirstDigitFound = 1;	// Ab der ersten Stelle, deren Wertigkeit größer 0 ist, müssen alle Werte übernommen werden
			*pText = (char)('0'+nHelpVal);	// Den Ascii-Wert der Wertigkeit in den String einfügen
			pText++;				// String-Pointer ein Zeichen weiterstellen

		}
		nValue = nValue % nDiff;		// Rest der Ganzzahldivision brint den Wert ohne die schon behandelte Stelle (für nächsten Durchlauf)
		nDiff = nDiff/10;				// Teiler um eine Stelle verringern (für nächsten Durchlauf)
	}
	// Die letzte Stelle wird immer eingefügt, für den Fall, daß der ganze Wert 0 ist.
	nHelpVal = nValue/nDiff;			// Ganzzahldivision bringt die Wertigkeit der letzten Stelle
	*pText = (char)('0'+nHelpVal);			// Den Ascii-Wert der Wertigkeit in den String einfügen
	pText++;						// String-Pointer ein Zeichen weiterstellen
	// String-Terminierung
	*pText = 0;
	return 0;
}

// NOLINTEND(readability-*, bugprone-easily-swappable-parameters, clang-diagnostic-invalid-utf8, clang-diagnostic-invalid-source-encoding, clang-diagnostic-pointer-arith, clang-diagnostic-strict-prototypes, hicpp-uppercase-literal-suffix, cppcoreguidelines-*, performance-*)
```

#### BrbAsciiToUdint.c - Wandelt einen String zu einem UDINT-Wert
```c
/********************************************************************
 * COPYRIGHT -- Bernecker + Rainer
 ********************************************************************
 * Library: BrbLib
 * File: BrbAsciiToUdint.c
 * Author: niedermeierr
 * Created: June 11, 2013
 ********************************************************************
 * Implementation of library BrbLib
 ********************************************************************/

#include <bur/plctypes.h>
#ifdef __cplusplus
	extern "C"
	{
#endif

#include "BrbLib.h"
#include <string.h>

#ifdef __cplusplus
	};
#endif

// NOLINTBEGIN(readability-*, bugprone-easily-swappable-parameters, clang-diagnostic-invalid-utf8, clang-diagnostic-invalid-source-encoding, clang-diagnostic-pointer-arith, clang-diagnostic-strict-prototypes, hicpp-uppercase-literal-suffix, cppcoreguidelines-*, performance-*)

/* Wandelt einen String zu einem UDINT-Wert */
unsigned long BrbAsciiToUdint(plcstring* pText)
{
	UDINT nFuncRetVal = 0;
	UDINT nCharCount = strlen((STRING*)pText )-1;
	STRING* pChar = 0;
	UDINT nDiff = 1; // Wertigkeit
	UDINT nDigitVal = 0; // Wert der Stelle als Einer-Wertigkeit
	while(1 == 1)
	{
		// Zeichen von hinten nach vorne durchlaufen
		pChar = (STRING*)pText+nCharCount;
		if(*pChar >= '0' && *pChar <= '9')
		{
			// Zeichen ist eine Nummer
			nDigitVal = (UDINT)(*pChar-'0'); // Wert als Einer-Stelle
			LREAL rResult = (LREAL)nFuncRetVal + ((LREAL)nDigitVal * (LREAL)nDiff);
			if(rResult > (LREAL)nBRB_UDINT_MAX)
			{
				// Ergebnis zu groß für UDINT
				nFuncRetVal = nBRB_UDINT_MAX; // Maximalen Wert zurückgeben
				break;
			}
			nFuncRetVal += nDigitVal * nDiff; // Wert als tatsächliche Wertigkeit zum Udint addieren
			nDiff *= 10; // Nächste Wertigkeit (Einer->Zehner->Hunderter->usw.)
		}
		else
		{
			// Zeichen ist keine Nummer -> Abbrechen
			break;
		}
		if(nCharCount > 0)
		{
			// Vorheriges Zeichen
			nCharCount--;
		}
		else
		{
			// Alle Zeichen durchlaufen
			break;
		}
	}
	return nFuncRetVal;
}

// NOLINTEND(readability-*, bugprone-easily-swappable-parameters, clang-diagnostic-invalid-utf8, clang-diagnostic-invalid-source-encoding, clang-diagnostic-pointer-arith, clang-diagnostic-strict-prototypes, hicpp-uppercase-literal-suffix, cppcoreguidelines-*, performance-*)
```

#### BrbUdintToHex.c - Wandelt einen Udint in einen Hex-String
```c
/********************************************************************
 * COPYRIGHT -- Bernecker + Rainer
 ********************************************************************
 * Library: BrbLib
 * File: BrbUdintToHex.c
 * Author: niedermeierr
 * Created: June 11, 2013
 ********************************************************************
 * Implementation of library BrbLib
 ********************************************************************/

#include <bur/plctypes.h>
#ifdef __cplusplus
	extern "C"
	{
#endif

#include "BrbLib.h"
#include <math.h>
#include <string.h>

#ifdef __cplusplus
	};
#endif

// NOLINTBEGIN(readability-*, bugprone-easily-swappable-parameters, clang-diagnostic-invalid-utf8, clang-diagnostic-invalid-source-encoding, clang-diagnostic-pointer-arith, clang-diagnostic-strict-prototypes, hicpp-uppercase-literal-suffix, cppcoreguidelines-*, performance-*)

/* Wandelt einen Udint in einen Hex-String */
unsigned short BrbUdintToHex(unsigned long nValue, plcstring* pHex, unsigned long nHexSize, plcbit bWithPraefix)
{
	memset(pHex, 0, nHexSize);
	if(bWithPraefix == 1)
	{
		BrbStringCat(pHex, "0x", nHexSize);
	}
	DINT nDigit = 0;
	for(nDigit=7; nDigit>=0; nDigit--)
	{
		UDINT nHelp1 = (UDINT)0xF << (UDINT)nDigit * 4;
		UDINT nHelp2 = nValue & nHelp1;
		UDINT nHelp3 = nHelp2 >> (UDINT)nDigit * 4;

		if(nHelp3 <= 9)
		{
			STRING sChar[2];
			sChar[0] = (char)('0' + nHelp3);
			sChar[1] = 0;
			BrbStringCat(pHex, sChar, nHexSize);
		}
		else
		{
			STRING sChar[2];
			sChar[0] = (char)('A' + nHelp3 - 10);
			sChar[1] = 0;
			BrbStringCat(pHex, sChar, nHexSize);
		}
	}
	return eBRB_ERR_OK;
}

// NOLINTEND(readability-*, bugprone-easily-swappable-parameters, clang-diagnostic-invalid-utf8, clang-diagnostic-invalid-source-encoding, clang-diagnostic-pointer-arith, clang-diagnostic-strict-prototypes, hicpp-uppercase-literal-suffix, cppcoreguidelines-*, performance-*)
```

#### BrbHexToUdint.c - Wandelt einen Hex-String in einen Udint
```c
/********************************************************************
 * COPYRIGHT -- Bernecker + Rainer
 ********************************************************************
 * Library: BrbLib
 * File: BrbHexToUdint.c
 * Author: niedermeierr
 * Created: June 11, 2013
 ********************************************************************
 * Implementation of library BrbLib
 ********************************************************************/

#include <bur/plctypes.h>
#ifdef __cplusplus
	extern "C"
	{
#endif

#include "BrbLib.h"
#include <math.h>
#include <string.h>

#ifdef __cplusplus
	};
#endif

// NOLINTBEGIN(readability-*, bugprone-easily-swappable-parameters, clang-diagnostic-invalid-utf8, clang-diagnostic-invalid-source-encoding, clang-diagnostic-pointer-arith, clang-diagnostic-strict-prototypes, hicpp-uppercase-literal-suffix, cppcoreguidelines-*, performance-*)

/* Wandelt einen Hex-String in einen Udint */
unsigned long BrbHexToUdint(plcstring* pHex)
{
	UDINT nResult = 0;
	UINT nBitDigit = 0;
	UDINT nHexLen = strlen((STRING*)pHex);
	DINT nCharIndex = 0;
	for(nCharIndex = (DINT)nHexLen-1; nCharIndex >= 0; nCharIndex--)
	{
		USINT* pChar = (USINT*)pHex+nCharIndex;
		UDINT nDigitValue = 0;
		LREAL rDigitValency = 0;
		if(*pChar >= 48 && *pChar <= 57)
		{
			nDigitValue = (*pChar-48);
		}
		else if(*pChar >= 65 && *pChar <= 70)
		{
			nDigitValue = (*pChar-55);
		}
		else if(*pChar >= 97 && *pChar <= 102)
		{
			nDigitValue = (*pChar-87);
		}
		rDigitValency = pow(2, nBitDigit);
		LREAL rResult = (LREAL)nResult + ((LREAL)nDigitValue * rDigitValency);
		if(rResult > (LREAL)nBRB_UDINT_MAX)
		{
			// Ergebnis zu groß für UDINT
			nResult = nBRB_UDINT_MAX; // Maximalen Wert zurückgeben
			break;
		}
		nResult = nResult + (nDigitValue * (UDINT)rDigitValency);
		nBitDigit += 4;
	}
	return nResult;
}

// NOLINTEND(readability-*, bugprone-easily-swappable-parameters, clang-diagnostic-invalid-utf8, clang-diagnostic-invalid-source-encoding, clang-diagnostic-pointer-arith, clang-diagnostic-strict-prototypes, hicpp-uppercase-literal-suffix, cppcoreguidelines-*, performance-*)
```

#### BrbUdintToBin.c - Wandelt einen Udint in einen Bin-String
```c
#include <bur/plctypes.h>
#ifdef __cplusplus
	extern "C"
	{
#endif

#include "BrbLib.h"
#include <math.h>
#include <string.h>

#ifdef __cplusplus
	};
#endif

// NOLINTBEGIN(readability-*, bugprone-easily-swappable-parameters, clang-diagnostic-invalid-utf8, clang-diagnostic-invalid-source-encoding, clang-diagnostic-pointer-arith, clang-diagnostic-strict-prototypes, hicpp-uppercase-literal-suffix, cppcoreguidelines-*, performance-*)

/* Wandelt einen Udint-Wert in einen Binär-String */
unsigned short BrbUdintToBin(unsigned long nValue, plcstring* pBin, unsigned long nBinSize, plcbit bWithPraefix)
{
	memset(pBin, 0, nBinSize);
	UDINT nCharIndex = 0;
	if(bWithPraefix == 1)
	{
		BrbStringCat(pBin, "%", nBinSize);
		nCharIndex += 1;
	}
	INT nBitNumber = 0;
	for(nBitNumber=31; nBitNumber>=0; nBitNumber--)
	{
		if(nCharIndex < nBinSize)
		{
			BOOL bBit = (nValue & ((UDINT)1 << nBitNumber)) > 0; // NOLINT(hicpp-signed-bitwise)
			if(bBit == 0)
			{
				*(pBin + nCharIndex) = 48;
			}
			else
			{
				*(pBin + nCharIndex) = 49;
			}
			nCharIndex++;
		}
		else
		{
			break;
		}
	}
	return 0;
}

// NOLINTEND(readability-*, bugprone-easily-swappable-parameters, clang-diagnostic-invalid-utf8, clang-diagnostic-invalid-source-encoding, clang-diagnostic-pointer-arith, clang-diagnostic-strict-prototypes, hicpp-uppercase-literal-suffix, cppcoreguidelines-*, performance-*)
```

#### BrbDintToHex.c - Wandelt eine DINT in einen Hex-String
```c
/********************************************************************
 * COPYRIGHT -- Bernecker + Rainer
 ********************************************************************
 * Library: BrbLib
 * File: BrbDintToHex.c
 * Author: niedermeierr
 * Created: January 17, 2017
 ********************************************************************
 * Implementation of library BrbLib
 ********************************************************************/

#include <bur/plctypes.h>
#ifdef __cplusplus
	extern "C"
	{
#endif

#include "BrbLib.h"
#include <math.h>
#include <string.h>

#ifdef __cplusplus
	};
#endif

// NOLINTBEGIN(readability-*, bugprone-easily-swappable-parameters, clang-diagnostic-invalid-utf8, clang-diagnostic-invalid-source-encoding, clang-diagnostic-pointer-arith, clang-diagnostic-strict-prototypes, hicpp-uppercase-literal-suffix, cppcoreguidelines-*, performance-*)

/* Wandelt einen DINT in einen Hex-String */
unsigned short BrbDintToHex(signed long nValue, plcstring* pHex, unsigned long nHexSize, plcbit bWithPraefix)
{
	// Die Bitmuster stimmen auch bei negativen Zahlen
	UDINT nValueUdint = (UDINT)nValue;
	BrbUdintToHex(nValueUdint, pHex, nHexSize, bWithPraefix);
	return 0;
}

// NOLINTEND(readability-*, bugprone-easily-swappable-parameters, clang-diagnostic-invalid-utf8, clang-diagnostic-invalid-source-encoding, clang-diagnostic-pointer-arith, clang-diagnostic-strict-prototypes, hicpp-uppercase-literal-suffix, cppcoreguidelines-*, performance-*)
```

#### BrbHexToDint.c - Wandelt einen Hex-String in einen Dint
```c
/********************************************************************
 * COPYRIGHT -- Bernecker + Rainer
 ********************************************************************
 * Library: BrbLib
 * File: BrbHexToDint.c
 * Author: niedermeierr
 * Created: January 19, 2017
 ********************************************************************
 * Implementation of library BrbLib
 ********************************************************************/

#include <bur/plctypes.h>
#ifdef __cplusplus
	extern "C"
	{
#endif

#include "BrbLib.h"
#include <math.h>
#include <string.h>

#ifdef __cplusplus
	};
#endif

// NOLINTBEGIN(readability-*, bugprone-easily-swappable-parameters, clang-diagnostic-invalid-utf8, clang-diagnostic-invalid-source-encoding, clang-diagnostic-pointer-arith, clang-diagnostic-strict-prototypes, hicpp-uppercase-literal-suffix, cppcoreguidelines-*, performance-*)

/* Wandelt einen Hex-String in einen Dint */
signed long BrbHexToDint(plcstring* pHex)
{
	DINT nResult = 0;
	UDINT nHexLen = strlen(pHex);
	UDINT nValueUdint = BrbHexToUdint(pHex);
	if(nHexLen < 8)
	{
		UDINT nMaxValuePositive = (UDINT)pow(2, nHexLen*4) - 1; // NOLINT(clang-diagnostic-bad-function-cast)
		UDINT nPolarityLimit = ((nMaxValuePositive+1) / 2) - 1;
		if(nValueUdint > nPolarityLimit)
		{
			// Zahl ist negativ
			nResult = (DINT)(nValueUdint - nMaxValuePositive - 1);
		}
		else
		{
			// Zahl ist positiv
			nResult = (DINT)nValueUdint;
		}
	}
	else
	{
		// Sonderbehandlung, weil die Berechnungen sonst durch Überlauf falsch wären
		if(nValueUdint > nBRB_DINT_MAX)
		{
			// Zahl ist negativ
			nResult = (DINT)(nValueUdint - nBRB_UDINT_MAX - 1);
		}
		else
		{
			// Zahl ist positiv
			nResult = (DINT)nValueUdint;
		}
	}
	return nResult;
}

// NOLINTEND(readability-*, bugprone-easily-swappable-parameters, clang-diagnostic-invalid-utf8, clang-diagnostic-invalid-source-encoding, clang-diagnostic-pointer-arith, clang-diagnostic-strict-prototypes, hicpp-uppercase-literal-suffix, cppcoreguidelines-*, performance-*)
```

#### BrbAsciiFieldToString.c - Wandelt ein Ascii-Feld in einen lesbaren String
```c
/********************************************************************
 * COPYRIGHT -- Bernecker + Rainer
 ********************************************************************
 * Library: BrbLib
 * File: BrbAsciiFieldToString.c
 * Author: niedermeierr
 * Created: April 04, 2014
 ********************************************************************
 * Implementation of library BrbLib
 ********************************************************************/

#include <bur/plctypes.h>
#ifdef __cplusplus
	extern "C"
	{
#endif

#include "BrbLib.h"
#include <string.h>

#ifdef __cplusplus
	};
#endif

// NOLINTBEGIN(readability-*, bugprone-easily-swappable-parameters, clang-diagnostic-invalid-utf8, clang-diagnostic-invalid-source-encoding, clang-diagnostic-pointer-arith, clang-diagnostic-strict-prototypes, hicpp-uppercase-literal-suffix, cppcoreguidelines-*, performance-*)

void AddCharText(USINT nAsciiChar, STRING* pText);

/* Wandelt ein Ascii-Feld in einen lesbaren Text */
plcbit BrbAsciiFieldToString(unsigned char* pAsciiField, unsigned long nAsciiFieldLen, unsigned long nFinalAsciiCharCount, plcstring* pText, unsigned long nTextSize) // NOLINT(readability-function-cognitive-complexity)
{
	BOOL bFuncRetVal = 0;
	if(pAsciiField != 0)
	{
		if(pText != 0)
		{
			// Textlänge für FinalAscii ermitteln
			if(nFinalAsciiCharCount > nAsciiFieldLen)
			{
				nFinalAsciiCharCount = nAsciiFieldLen;
			}
			UDINT nFinalAsciiTextLen = 0;
			if(nFinalAsciiCharCount > 0)
			{
				// Letzte Zeichenanzahl solange vermindern, bis übersetzter FinalText in pText passt
				BOOL bTextSizeToSmall = 0;
				DINT nIndex = 0;
				for(nIndex=(DINT)nFinalAsciiCharCount; nIndex>0; nIndex--)
				{
					USINT* pFinalAsciiBegin = pAsciiField + nAsciiFieldLen - nFinalAsciiCharCount;
					bTextSizeToSmall = BrbAsciiFieldToString(pFinalAsciiBegin, nFinalAsciiCharCount, 0, pText, nTextSize);
					nFinalAsciiTextLen = strlen(pText);
					if(bTextSizeToSmall == 0)
					{
						// Übersetzter FinalText passt in pText
						break;
					}
					nFinalAsciiCharCount--;
				}
				if(bTextSizeToSmall == 1)
				{
					// Auch das letzte Zeichen passt übersetzt nicht in pText
					nFinalAsciiCharCount = 0;
					nFinalAsciiTextLen = 0;
				}
			}
			memset((STRING*)pText, 0, nTextSize);
			UDINT nAsciiFieldIndex = 0;
			USINT* pAsciiChar = 0;
			DINT nTextIndex = 0;
			STRING sCharDescription[30];
			STRING sCharDescriptionStart[5];
			strcpy(sCharDescriptionStart, "<");
			STRING sCharDescriptionEnd[5];
			strcpy(sCharDescriptionEnd, ">");
			UDINT nCharDescriptionLen = 0;
			// Platz vorsehen für die letzten Ascii-Zeichen und Platzhalter
			DINT nPlaceHolderLen = 7; // "<+9999>"
			DINT nTextLimit = (DINT)nTextSize - (DINT)nFinalAsciiTextLen - nPlaceHolderLen - 1;
			BOOL bTextOverrun = 0;
			BOOL bHandleFinalAscii = 0;
			BOOL bLeave = 0;
			do
			{
				pAsciiChar = ((USINT*)pAsciiField) + nAsciiFieldIndex;
				if(*pAsciiChar < 32)
				{
					// Sonderzeichen -> Anzahl dieses Sonderzeichens zählen
					USINT* pAsciiCharPreview = 0;
					UDINT nSameAsciiCharCount = 1;
					for(pAsciiCharPreview=pAsciiChar+1; pAsciiCharPreview<=pAsciiField+nAsciiFieldLen-1; pAsciiCharPreview++)
					{
						if(*pAsciiCharPreview == *pAsciiChar)
						{
							nSameAsciiCharCount++;
						}
						else
						{
							break;
						}
					}
					if(nSameAsciiCharCount == 1)
					{
						// Zeichen kommt nur einmal vor
						memset(sCharDescription, 0, sizeof(sCharDescription));
						BrbStringCat(sCharDescription, sCharDescriptionStart, sizeof(sCharDescription));
						AddCharText(*pAsciiChar, sCharDescription);
						BrbStringCat(sCharDescription, sCharDescriptionEnd, sizeof(sCharDescription));
						nCharDescriptionLen = strlen(sCharDescription);
						if(nTextIndex < nTextLimit-(DINT)nCharDescriptionLen)
						{
							BrbStringCat(pText, sCharDescription, nTextSize);
							nTextIndex += (DINT)nCharDescriptionLen;
							nAsciiFieldIndex += 1;
						}
						else
						{
							bTextOverrun = 1;
							bFuncRetVal = 1;
						}
					}
					else
					{
						// Zeichen kommt öfters vor
						memset(sCharDescription, 0, sizeof(sCharDescription));
						BrbStringCat(sCharDescription, sCharDescriptionStart, sizeof(sCharDescription));
						STRING sItoa[10];
						memset(sItoa, 0, sizeof(sItoa));
						BrbUdintToAscii(nSameAsciiCharCount, sItoa);
						BrbStringCat(sCharDescription, sItoa, sizeof(sCharDescription));
						BrbStringCat(sCharDescription, "*", sizeof(sCharDescription));
						AddCharText(*pAsciiChar, sCharDescription);
						BrbStringCat(sCharDescription, sCharDescriptionEnd, sizeof(sCharDescription));
						nCharDescriptionLen = strlen(sCharDescription);
						if(nTextIndex < nTextLimit-(DINT)nCharDescriptionLen)
						{
							BrbStringCat(pText, sCharDescription, nTextSize);
							nTextIndex += (DINT)nCharDescriptionLen;
							nAsciiFieldIndex += nSameAsciiCharCount;
						}
						else
						{
							bTextOverrun = 1;
							bFuncRetVal = 1;
						}
					}
				}
				else
				{
					// Normalzeichen -> übernehmen
					if(nTextIndex < nTextLimit-1)
					{
						USINT* pTextChar = ((USINT*)pText) + nTextIndex;
						*pTextChar = *pAsciiChar;
						nTextIndex++;
						nAsciiFieldIndex += 1;
					}
					else
					{
						bTextOverrun = 1;
						bFuncRetVal = 1;
					}
				}
				if(bTextOverrun == 1 || nAsciiFieldIndex >= (nAsciiFieldLen-nFinalAsciiCharCount))
				{
					if(bHandleFinalAscii == 0 && nFinalAsciiCharCount > 0)
					{
						// Die letzten Zeichen müssen enthalten sein (Platz im Text dafür wurde vorgesehen)
						DINT nPlaceholderCharCount = (DINT)nAsciiFieldLen - (DINT)nAsciiFieldIndex - (DINT)nFinalAsciiCharCount;
						if(nPlaceholderCharCount > 0)
						{
							STRING sPlaceholder[10];
							memset(sPlaceholder, 0, sizeof(sPlaceholder));
							BrbStringCat(sPlaceholder, "<+", sizeof(sPlaceholder));
							STRING sItoa[10];
							memset(sItoa, 0, sizeof(sItoa));
							brsitoa((DINT)nPlaceholderCharCount, (UDINT)&sItoa);
							BrbStringCat(sPlaceholder, sItoa, sizeof(sPlaceholder));
							BrbStringCat(sPlaceholder, ">", sizeof(sPlaceholder));
							BrbStringCat(pText, sPlaceholder, nTextSize);
							nTextIndex += (DINT)strlen(sPlaceholder);
						}
						nTextLimit = (DINT)nTextSize - 1;
						bTextOverrun = 0;
						if(nAsciiFieldIndex < nAsciiFieldLen - nFinalAsciiCharCount)
						{
							nAsciiFieldIndex = nAsciiFieldLen - nFinalAsciiCharCount;
						}
						bHandleFinalAscii = 1;
						bLeave = 0;
					}
					else if(nFinalAsciiCharCount == 0)
					{
						// Es gibt keine Finalzeichen -> Anzahl der austehenden Zeichen schreiben und beenden
						DINT nPlaceholderCharCount = (DINT)nAsciiFieldLen - (DINT)nAsciiFieldIndex;
						if(nPlaceholderCharCount > 0)
						{
							STRING sPlaceholder[10];
							memset(sPlaceholder, 0, sizeof(sPlaceholder));
							BrbStringCat(sPlaceholder, "<+", sizeof(sPlaceholder));
							STRING sItoa[10];
							memset(sItoa, 0, sizeof(sItoa));
							brsitoa((DINT)nPlaceholderCharCount, (UDINT)&sItoa);
							BrbStringCat(sPlaceholder, sItoa, sizeof(sPlaceholder));
							BrbStringCat(sPlaceholder, ">", sizeof(sPlaceholder));
							BrbStringCat(pText, sPlaceholder, nTextSize);
							nTextIndex += (DINT)strlen(sPlaceholder);
						}
						bLeave =1;
					}
				}
				if(nAsciiFieldIndex >= nAsciiFieldLen)
				{
					// Ende des Ascii-Feldes erreicht
					bLeave = 1;
				}
			} while(bLeave == 0);
		}
	}
	return bFuncRetVal;
}

void AddCharText(USINT nAsciiChar, STRING* pText) // NOLINT(readability-function-cognitive-complexity)
{
	// NOLINTBEGIN(clang-analyzer-security.insecureAPI.strcpy)
	if(nAsciiChar == 0)
	{
		strcat(pText, "0=NUL");
	}
	else if(nAsciiChar == 1)
	{
		strcat(pText, "1=SOH");
	}
	else if(nAsciiChar == 2)
	{
		strcat(pText, "2=STX");
	}
	else if(nAsciiChar == 3)
	{
		strcat(pText, "3=ETX");
	}
	else if(nAsciiChar == 4)
	{
		strcat(pText, "4=EOT");
	}
	else if(nAsciiChar == 5)
	{
		strcat(pText, "5=ENQ");
	}
	else if(nAsciiChar == 6)
	{
		strcat(pText, "6=ACK");
	}
	else if(nAsciiChar == 7)
	{
		strcat(pText, "7=BEL");
	}
	else if(nAsciiChar == 8)
	{
		strcat(pText, "8=BS");
	}
	else if(nAsciiChar == 9)
	{
		strcat(pText, "9=HT");
	}
	else if(nAsciiChar == 10)
	{
		strcat(pText, "10=LF");
	}
	else if(nAsciiChar == 11)
	{
		strcat(pText, "11=VT");
	}
	else if(nAsciiChar == 12)
	{
		strcat(pText, "12=FF");
	}
	else if(nAsciiChar == 13)
	{
		strcat(pText, "13=CR");
	}
	else if(nAsciiChar == 14)
	{
		strcat(pText, "14=SO");
	}
	else if(nAsciiChar == 15)
	{
		strcat(pText, "15=SI");
	}
	else if(nAsciiChar == 16)
	{
		strcat(pText, "16=DL");
	}
	else if(nAsciiChar == 17)
	{
		strcat(pText, "17=DC");
	}
	else if(nAsciiChar == 18)
	{
		strcat(pText, "18=DC2");
	}
	else if(nAsciiChar == 19)
	{
		strcat(pText, "19=DC3");
	}
	else if(nAsciiChar == 20)
	{
		strcat(pText, "20=DC4");
	}
	else if(nAsciiChar == 21)
	{
		strcat(pText, "21=NAK");
	}
	else if(nAsciiChar == 22)
	{
		strcat(pText, "22=SYN");
	}
	else if(nAsciiChar == 23)
	{
		strcat(pText, "23=ETB");
	}
	else if(nAsciiChar == 24)
	{
		strcat(pText, "24=CAN");
	}
	else if(nAsciiChar == 25)
	{
		strcat(pText, "25=EM");
	}
	else if(nAsciiChar == 26)
	{
		strcat(pText, "26=SUB");
	}
	else if(nAsciiChar == 27)
	{
		strcat(pText, "27=ESC");
	}
	else if(nAsciiChar == 28)
	{
		strcat(pText, "28=FS");
	}
	else if(nAsciiChar == 29)
	{
		strcat(pText, "29=GS");
	}
	else if(nAsciiChar == 30)
	{
		strcat(pText, "30=RS");
	}
	else if(nAsciiChar == 31)
	{
		strcat(pText, "31=US");
	}
	else
	{
		STRING sItoa[10];
		memset(sItoa, 0, sizeof(sItoa));
		brsitoa((DINT)nAsciiChar, (UDINT)&sItoa);
		strcat(pText, sItoa);
	}
	// NOLINTEND(clang-analyzer-security.insecureAPI.strcpy)
}

// NOLINTEND(readability-*, bugprone-easily-swappable-parameters, clang-diagnostic-invalid-utf8, clang-diagnostic-invalid-source-encoding, clang-diagnostic-pointer-arith, clang-diagnostic-strict-prototypes, hicpp-uppercase-literal-suffix, cppcoreguidelines-*, performance-*)
```

#### BrbStringGetIndexOf.c - Gibt den Index einer Zeichenfolge innerhalb einesTextes zurück
```c
/********************************************************************
 * COPYRIGHT -- Bernecker + Rainer
 ********************************************************************
 * Library: BrbLib
 * File: BrbStringGetIndexOf.c
 * Author: niedermeierr
 * Created: June 11, 2013
 ********************************************************************
 * Implementation of library BrbLib
 ********************************************************************/

#include <bur/plctypes.h>
#ifdef __cplusplus
	extern "C"
	{
#endif

#include "BrbLib.h"
#include <string.h>

#ifdef __cplusplus
	};
#endif

// NOLINTBEGIN(readability-*, bugprone-easily-swappable-parameters, clang-diagnostic-invalid-utf8, clang-diagnostic-invalid-source-encoding, clang-diagnostic-pointer-arith, clang-diagnostic-strict-prototypes, hicpp-uppercase-literal-suffix, cppcoreguidelines-*, performance-*)

/* Gibt den ersten Index eines zu suchenden Textes zurück */
signed long BrbStringGetIndexOf(plcstring* pText, plcstring* pFind, unsigned long nTextLen)
{
	DINT nResult = -1;
	// Wenn die Länge bekannt ist, kann sie übergeben werden
	// Damit entfällt das Aufrufen von strlen, welches bei langen Texten Zeit braucht
	UDINT nLenText = nTextLen;
	if(nTextLen == 0)
	{
		nLenText = strlen(pText);
	}
	UDINT nLenFind = strlen(pFind);
	UDINT nCharIndex = 0;
	// Text von vorne nach hinten durchsuchen
	for(nCharIndex=0; nCharIndex<nLenText; nCharIndex++)
	{
		// Textstelle vergleichen
		if(memcmp((pText + nCharIndex), pFind, nLenFind) == 0)
		{
			// Text gefunden
			nResult = (DINT)nCharIndex;
			break;
		}
	}
	return nResult;
}

// NOLINTEND(readability-*, bugprone-easily-swappable-parameters, clang-diagnostic-invalid-utf8, clang-diagnostic-invalid-source-encoding, clang-diagnostic-pointer-arith, clang-diagnostic-strict-prototypes, hicpp-uppercase-literal-suffix, cppcoreguidelines-*, performance-*)
```

#### BrbStringGetLastIndexOf.c - Gibt den letzten Index einer Zeichenfolge innerhalb einesTextes zurück
```c
/********************************************************************
 * COPYRIGHT -- Bernecker + Rainer
 ********************************************************************
 * Library: BrbLib
 * File: BrbStringGetLastIndexOf.c
 * Author: niedermeierr
 * Created: December 01, 2014
 *******************************************************************/

#include <bur/plctypes.h>
#ifdef __cplusplus
	extern "C"
	{
#endif

#include "BrbLib.h"
#include <string.h>

#ifdef __cplusplus
	};
#endif

// NOLINTBEGIN(readability-*, bugprone-easily-swappable-parameters, clang-diagnostic-invalid-utf8, clang-diagnostic-invalid-source-encoding, clang-diagnostic-pointer-arith, clang-diagnostic-strict-prototypes, hicpp-uppercase-literal-suffix, cppcoreguidelines-*, performance-*)

/* Gibt den letzten Index eines zu suchenden Textes zurück */
signed long BrbStringGetLastIndexOf(plcstring* pText, plcstring* pFind, unsigned long nTextLen)
{
	DINT nResult = -1;
	// Wenn die Länge bekannt ist, kann sie übergeben werden
	// Damit entfällt das Aufrufen von strlen, welches bei langen Texten Zeit braucht
	UDINT nLenText = nTextLen;
	if(nTextLen == 0)
	{
		nLenText = strlen(pText);
	}
	UDINT nLenFind = strlen(pFind);
	DINT nCharIndex = 0;
	// Text von hinten nach vorne durchsuchen
	for(nCharIndex=(DINT)nLenText-1; nCharIndex>=0; nCharIndex--)
	{
		// Textstelle vergleichen
		if(memcmp((pText + nCharIndex), pFind, nLenFind) == 0)
		{
			// Text gefunden
			nResult = nCharIndex;
			break;
		}
	}
	return nResult;
}

// NOLINTEND(readability-*, bugprone-easily-swappable-parameters, clang-diagnostic-invalid-utf8, clang-diagnostic-invalid-source-encoding, clang-diagnostic-pointer-arith, clang-diagnostic-strict-prototypes, hicpp-uppercase-literal-suffix, cppcoreguidelines-*, performance-*)
```

#### BrbStringGetAdrOf.c - Gibt die Adresse eines zu suchenden Textes zurück
```c
/********************************************************************
 * COPYRIGHT -- Bernecker + Rainer
 ********************************************************************
 * Library: BrbLib
 * File: BrbStringGetAdrOf.c
 * Author: niedermeierr
 * Created: June 11, 2013
 ********************************************************************
 * Implementation of library BrbLib
 ********************************************************************/

#include <bur/plctypes.h>
#ifdef __cplusplus
	extern "C"
	{
#endif

#include "BrbLib.h"
#include <string.h>

#ifdef __cplusplus
	};
#endif

// NOLINTBEGIN(readability-*, bugprone-easily-swappable-parameters, clang-diagnostic-invalid-utf8, clang-diagnostic-invalid-source-encoding, clang-diagnostic-pointer-arith, clang-diagnostic-strict-prototypes, hicpp-uppercase-literal-suffix, cppcoreguidelines-*, performance-*)

/* Gibt die erste Adresse eines zu suchenden Textes zurück */
plcstring* BrbStringGetAdrOf(plcstring* pText, plcstring* pFind, unsigned long nTextLen)
{
	STRING* pResult = 0;
	// Wenn die Länge bekannt ist, kann sie übergeben werden
	// Damit entfällt das Aufrufen von strlen, welches bei langen Texten Zeit braucht
	UDINT nLenText = nTextLen;
	if(nTextLen == 0)
	{
		nLenText = strlen(pText);
	}
	UDINT nLenFind = strlen(pFind);
	UDINT nCharIndex = 0;
	// Text von vorne nach hinten durchsuchen
	for(nCharIndex=0; nCharIndex<nLenText; nCharIndex++)
	{
		// Textstelle vergleichen
		if(memcmp((pText + nCharIndex), pFind, nLenFind) == 0)
		{
			// Text gefunden
			pResult = pText + nCharIndex;
			break;
		}
	}
	return pResult;
}

// NOLINTEND(readability-*, bugprone-easily-swappable-parameters, clang-diagnostic-invalid-utf8, clang-diagnostic-invalid-source-encoding, clang-diagnostic-pointer-arith, clang-diagnostic-strict-prototypes, hicpp-uppercase-literal-suffix, cppcoreguidelines-*, performance-*)
```

#### BrbStringGetLastAdrOf.c - Gibt die letzte Adresse eines zu suchenden Textes zurück
```c
/********************************************************************
 * COPYRIGHT -- Bernecker + Rainer
 ********************************************************************
 * Library: BrbLib
 * File: BrbStringGetLastAdrOf.c
 * Author: niedermeierr
 * Created: October 21, 2014
 ********************************************************************
 * Implementation of library BrbLib
 ********************************************************************/

#include <bur/plctypes.h>
#ifdef __cplusplus
	extern "C"
	{
#endif

#include "BrbLib.h"
#include <string.h>

#ifdef __cplusplus
	};
#endif

// NOLINTBEGIN(readability-*, bugprone-easily-swappable-parameters, clang-diagnostic-invalid-utf8, clang-diagnostic-invalid-source-encoding, clang-diagnostic-pointer-arith, clang-diagnostic-strict-prototypes, hicpp-uppercase-literal-suffix, cppcoreguidelines-*, performance-*)

/* Gibt die letzte Adresse eines zu suchenden Textes zurück */
plcstring* BrbStringGetLastAdrOf(plcstring* pText, plcstring* pFind, unsigned long nTextLen)
{
	STRING* pResult = 0;
	// Wenn die Länge bekannt ist, kann sie übergeben werden
	// Damit entfällt das Aufrufen von strlen, welches bei langen Texten Zeit braucht
	UDINT nLenText = nTextLen;
	if(nTextLen == 0)
	{
		nLenText = strlen(pText);
	}
	UDINT nLenFind = strlen(pFind);
	DINT nCharIndex = 0;
	// Text von hinten nach vorne durchsuchen
	for(nCharIndex=(DINT)nLenText-1; nCharIndex>=0; nCharIndex--)
	{
		// Textstelle vergleichen
		if(memcmp((pText + nCharIndex), pFind, nLenFind) == 0)
		{
			// Text gefunden
			pResult = pText + nCharIndex;
			break;
		}
	}
	return pResult;
}

// NOLINTEND(readability-*, bugprone-easily-swappable-parameters, clang-diagnostic-invalid-utf8, clang-diagnostic-invalid-source-encoding, clang-diagnostic-pointer-arith, clang-diagnostic-strict-prototypes, hicpp-uppercase-literal-suffix, cppcoreguidelines-*, performance-*)
```

#### BrbStringStartsWith.c - Gibt zurück, ob ein Text mit einer bestimmten Zeichenfolge beginnt
```c
/********************************************************************
 * COPYRIGHT -- Bernecker + Rainer
 ********************************************************************
 * Library: BrbLib
 * File: BrbStringStartsWith.c
 * Author: niedermeierr
 * Created: June 11, 2013
 ********************************************************************
 * Implementation of library BrbLib
 ********************************************************************/

#include <bur/plctypes.h>
#ifdef __cplusplus
	extern "C"
	{
#endif

#include "BrbLib.h"
#include <string.h>

#ifdef __cplusplus
	};
#endif

// NOLINTBEGIN(readability-*, bugprone-easily-swappable-parameters, clang-diagnostic-invalid-utf8, clang-diagnostic-invalid-source-encoding, clang-diagnostic-pointer-arith, clang-diagnostic-strict-prototypes, hicpp-uppercase-literal-suffix, cppcoreguidelines-*, performance-*)

/* Gibt zurück, ob ein Text mit einer bestimmten Zeichenfolge beginnt */
plcbit BrbStringStartsWith(plcstring* pText, plcstring* pFind)
{
	BOOL bResult = 0;
	UDINT nLenFind = strlen(pFind);
	if(memcmp(pText, pFind, nLenFind) == 0)
	{
		bResult = 1;
	}
	return bResult;
}

// NOLINTEND(readability-*, bugprone-easily-swappable-parameters, clang-diagnostic-invalid-utf8, clang-diagnostic-invalid-source-encoding, clang-diagnostic-pointer-arith, clang-diagnostic-strict-prototypes, hicpp-uppercase-literal-suffix, cppcoreguidelines-*, performance-*)
```

#### BrbStringEndsWith.c - Gibt zurück, ob ein Text mit einer bestimmten Zeichenfolge endet
```c
/********************************************************************
 * COPYRIGHT -- Bernecker + Rainer
 ********************************************************************
 * Library: BrbLib
 * File: BrbStringEndsWith.c
 * Author: niedermeierr
 * Created: June 11, 2013
 ********************************************************************
 * Implementation of library BrbLib
 ********************************************************************/

#include <bur/plctypes.h>
#ifdef __cplusplus
	extern "C"
	{
#endif

#include "BrbLib.h"
#include <string.h>

#ifdef __cplusplus
	};
#endif

// NOLINTBEGIN(readability-*, bugprone-easily-swappable-parameters, clang-diagnostic-invalid-utf8, clang-diagnostic-invalid-source-encoding, clang-diagnostic-pointer-arith, clang-diagnostic-strict-prototypes, hicpp-uppercase-literal-suffix, cppcoreguidelines-*, performance-*)

/* Gibt zurück, ob ein Text mit einer bestimmten Zeichenfolge endet */
plcbit BrbStringEndsWith(plcstring* pText, plcstring* pFind)
{
	BOOL bResult = 0;
	UDINT nLenText = strlen(pText);
	UDINT nLenFind = strlen(pFind);
	if(nLenText >= nLenFind)
	{
		if(memcmp(pText + nLenText - nLenFind, pFind, nLenFind) == 0)
		{
			bResult = 1;
		}
	}
	return bResult;
}

// NOLINTEND(readability-*, bugprone-easily-swappable-parameters, clang-diagnostic-invalid-utf8, clang-diagnostic-invalid-source-encoding, clang-diagnostic-pointer-arith, clang-diagnostic-strict-prototypes, hicpp-uppercase-literal-suffix, cppcoreguidelines-*, performance-*)
```

#### BrbStringGetSubText.c - Gibt eine Zeichenfolge innerhalb eines Textes zurück
```c
/********************************************************************
 * COPYRIGHT -- Bernecker + Rainer
 ********************************************************************
 * Library: BrbLib
 * File: BrbStringGetSubText.c
 * Author: niedermeierr
 * Created: July 05, 2013
 ********************************************************************
 * Implementation of library BrbLib
 ********************************************************************/

#include <bur/plctypes.h>
#ifdef __cplusplus
	extern "C"
	{
#endif

#include "BrbLib.h"
#include <string.h>

#ifdef __cplusplus
	};
#endif

// NOLINTBEGIN(readability-*, bugprone-easily-swappable-parameters, clang-diagnostic-invalid-utf8, clang-diagnostic-invalid-source-encoding, clang-diagnostic-pointer-arith, clang-diagnostic-strict-prototypes, hicpp-uppercase-literal-suffix, cppcoreguidelines-*, performance-*)

/* Gibt eine Zeichenfolge innerhalb eines Textes zurück */
plcstring* BrbStringGetSubText(plcstring* pText, unsigned long nIndex, unsigned long nLen, plcstring* pSubText)
{
	memcpy(pSubText, (pText + nIndex), nLen);
	pSubText[nLen] = 0; // NullTerminierung
	return (STRING*)(pText + nIndex + nLen);
}

// NOLINTEND(readability-*, bugprone-easily-swappable-parameters, clang-diagnostic-invalid-utf8, clang-diagnostic-invalid-source-encoding, clang-diagnostic-pointer-arith, clang-diagnostic-strict-prototypes, hicpp-uppercase-literal-suffix, cppcoreguidelines-*, performance-*)
```

#### BrbStringGetSubTextByLen.c - Gibt eine Zeichenfolge innerhalb eines Textes zurück
```c
/********************************************************************
 * COPYRIGHT -- Bernecker + Rainer
 ********************************************************************
 * Library: BrbLib
 * File: BrbStringGetSubTextByLen.c
 * Author: niedermeierr
 * Created: June 17, 2013
 ********************************************************************
 * Implementation of library BrbLib
 ********************************************************************/

#include <bur/plctypes.h>
#ifdef __cplusplus
	extern "C"
	{
#endif

#include "BrbLib.h"
#include <string.h>

#ifdef __cplusplus
	};
#endif

// NOLINTBEGIN(readability-*, bugprone-easily-swappable-parameters, clang-diagnostic-invalid-utf8, clang-diagnostic-invalid-source-encoding, clang-diagnostic-pointer-arith, clang-diagnostic-strict-prototypes, hicpp-uppercase-literal-suffix, cppcoreguidelines-*, performance-*)

/* Gibt eine Zeichenfolge innerhalb eines Textes zurück */
plcstring* BrbStringGetSubTextByLen(plcstring* pStart, unsigned long nLen, plcstring* pSubText)
{
	memcpy(pSubText, pStart, nLen);
	pSubText[nLen] = 0; // NullTerminierung
	return (STRING*)(pStart + nLen);
}

// NOLINTEND(readability-*, bugprone-easily-swappable-parameters, clang-diagnostic-invalid-utf8, clang-diagnostic-invalid-source-encoding, clang-diagnostic-pointer-arith, clang-diagnostic-strict-prototypes, hicpp-uppercase-literal-suffix, cppcoreguidelines-*, performance-*)
```

#### BrbStringGetSubTextByAdr.c - Gibt eine Zeichenfolge innerhalb eines Textes zurück
```c
/********************************************************************
 * COPYRIGHT -- Bernecker + Rainer
 ********************************************************************
 * Library: BrbLib
 * File: BrbStringGetSubTextByAdr.c
 * Author: niedermeierr
 * Created: June 17, 2013
 ********************************************************************
 * Implementation of library BrbLib
 ********************************************************************/

#include <bur/plctypes.h>
#ifdef __cplusplus
	extern "C"
	{
#endif

#include "BrbLib.h"
#include <string.h>

#ifdef __cplusplus
	};
#endif

// NOLINTBEGIN(readability-*, bugprone-easily-swappable-parameters, clang-diagnostic-invalid-utf8, clang-diagnostic-invalid-source-encoding, clang-diagnostic-pointer-arith, clang-diagnostic-strict-prototypes, hicpp-uppercase-literal-suffix, cppcoreguidelines-*, performance-*)

/* Gibt eine Zeichenfolge innerhalb eines Textes zurück */
plcstring* BrbStringGetSubTextByAdr(plcstring* pStart, plcstring* pEnd, plcstring* pSubText)
{
	STRING* pResult = 0;
	if(pEnd > pStart)
	{
		UDINT nLen = (UDINT)pEnd - (UDINT)pStart;
		pResult = BrbStringGetSubTextByLen(pStart, nLen, pSubText);
	}
	return pResult;
}

// NOLINTEND(readability-*, bugprone-easily-swappable-parameters, clang-diagnostic-invalid-utf8, clang-diagnostic-invalid-source-encoding, clang-diagnostic-pointer-arith, clang-diagnostic-strict-prototypes, hicpp-uppercase-literal-suffix, cppcoreguidelines-*, performance-*)
```

#### BrbStringAppend.c - Hängt eine Zeichenfolge an einen Text (Ersatz für strcat)
```c
/********************************************************************
 * COPYRIGHT -- Bernecker + Rainer
 ********************************************************************
 * Library: BrbLib
 * File: BrbStringAppend.c
 * Author: niedermeierr
 * Created: February 17, 2016
 ********************************************************************
 * Implementation of library BrbLib
 ********************************************************************/

#include <bur/plctypes.h>
#ifdef __cplusplus
	extern "C"
	{
#endif

#include "BrbLib.h"
#include <string.h>

#ifdef __cplusplus
	};
#endif

// NOLINTBEGIN(readability-*, bugprone-easily-swappable-parameters, clang-diagnostic-invalid-utf8, clang-diagnostic-invalid-source-encoding, clang-diagnostic-pointer-arith, clang-diagnostic-strict-prototypes, hicpp-uppercase-literal-suffix, cppcoreguidelines-*, performance-*)

/* Hängt eine Zeichenfolge an einen Text (Ersatz für strcat) */
unsigned long BrbStringAppend(plcstring* pText, plcstring* pTextAppend, unsigned long* pTextOffset)
{
	UDINT nAppendLen = strlen(pTextAppend);
	memcpy(pText + *pTextOffset, pTextAppend, nAppendLen);
	*pTextOffset += nAppendLen;
	*(pText + *pTextOffset) = 0; // String-Abschluss
	return nAppendLen;
}

// NOLINTEND(readability-*, bugprone-easily-swappable-parameters, clang-diagnostic-invalid-utf8, clang-diagnostic-invalid-source-encoding, clang-diagnostic-pointer-arith, clang-diagnostic-strict-prototypes, hicpp-uppercase-literal-suffix, cppcoreguidelines-*, performance-*)
```

#### BrbStringCut.c - Schneidet eine Zeichenfolge aus einem Text heraus
```c
/********************************************************************
 * COPYRIGHT -- Bernecker + Rainer
 ********************************************************************
 * Library: BrbLib
 * File: BrbStringCut.c
 * Author: niedermeierr
 * Created: July 05, 2013
 ********************************************************************
 * Implementation of library BrbLib
 ********************************************************************/

#include <bur/plctypes.h>
#ifdef __cplusplus
	extern "C"
	{
#endif

#include "BrbLib.h"
#include <string.h>

#ifdef __cplusplus
	};
#endif

// NOLINTBEGIN(readability-*, bugprone-easily-swappable-parameters, clang-diagnostic-invalid-utf8, clang-diagnostic-invalid-source-encoding, clang-diagnostic-pointer-arith, clang-diagnostic-strict-prototypes, hicpp-uppercase-literal-suffix, cppcoreguidelines-*, performance-*)

/* Schneidet eine Zeichenfolge aus einem Text heraus */
plcstring* BrbStringCut(plcstring* pText, unsigned long nCutIndex, unsigned long nCutLen, plcstring* pCut)
{
	STRING* pResult = 0;
	UDINT nTextLen = strlen(pText);
	if(nCutIndex+nCutLen > nTextLen)
	{
		nCutLen = nTextLen-nCutIndex;
	}
	UDINT nRestLen = nTextLen - nCutIndex - nCutLen + 1;
	if(pCut != 0)
	{
		// Herauszuschneidenden String kopieren
		memcpy(pCut, (pText + nCutIndex), nCutLen);
		*(pCut + nCutLen) = 0;
	}
	// Zeichen nach dem Cut nach vorne ziehen
	memmove((pText + nCutIndex), (pText + nCutIndex + nCutLen), nRestLen);
	pResult = pText + nCutIndex + nCutLen;
	return pResult;
}

// NOLINTEND(readability-*, bugprone-easily-swappable-parameters, clang-diagnostic-invalid-utf8, clang-diagnostic-invalid-source-encoding, clang-diagnostic-pointer-arith, clang-diagnostic-strict-prototypes, hicpp-uppercase-literal-suffix, cppcoreguidelines-*, performance-*)
```

#### BrbStringCutFromLastSeparator.c - Schneidet die Zeichenfolge ab dem letzten Trennzeichen in einem Text ab
```c
/********************************************************************
 * COPYRIGHT -- Bernecker + Rainer
 ********************************************************************
 * Library: BrbLib
 * File: BrbStringCutFromLastSeparator.c
 * Author: niedermeierr
 * Created: October 21, 2014
 ********************************************************************
 * Implementation of library BrbLib
 ********************************************************************/

#include <bur/plctypes.h>
#ifdef __cplusplus
	extern "C"
	{
#endif

#include "BrbLib.h"
#include <string.h>

#ifdef __cplusplus
	};
#endif

// NOLINTBEGIN(readability-*, bugprone-easily-swappable-parameters, clang-diagnostic-invalid-utf8, clang-diagnostic-invalid-source-encoding, clang-diagnostic-pointer-arith, clang-diagnostic-strict-prototypes, hicpp-uppercase-literal-suffix, cppcoreguidelines-*, performance-*)

/* Schneidet die Zeichenfolge ab dem letzten Trennzeichen in einem Text ab */
unsigned long BrbStringCutFromLastSeparator(plcstring* pText, plcstring* pSeparator, plcstring* pCut)
{
	UDINT nResult = 0;
	UDINT nTextLen = strlen(pText);
	STRING* pSeparatorStart = BrbStringGetLastAdrOf(pText, pSeparator, nTextLen);
	if(pSeparatorStart != 0)
	{
		UDINT nCutIndex = (UDINT)(pSeparatorStart - pText);
		UDINT nCutLen = nTextLen - nCutIndex;
		BrbStringCut(pText, nCutIndex, nCutLen, pCut);
		nResult = nCutLen;
	}
	return nResult;
}

// NOLINTEND(readability-*, bugprone-easily-swappable-parameters, clang-diagnostic-invalid-utf8, clang-diagnostic-invalid-source-encoding, clang-diagnostic-pointer-arith, clang-diagnostic-strict-prototypes, hicpp-uppercase-literal-suffix, cppcoreguidelines-*, performance-*)
```

#### BrbStringInsert.c - Fügt eine Zeichenfolge in einen Text ein
```c
/********************************************************************
 * COPYRIGHT -- Bernecker + Rainer
 ********************************************************************
 * Library: BrbLib
 * File: BrbStringInsert.c
 * Author: niedermeierr
 * Created: July 05, 2013
 ********************************************************************
 * Implementation of library BrbLib
 ********************************************************************/

#include <bur/plctypes.h>
#ifdef __cplusplus
	extern "C"
	{
#endif

#include "BrbLib.h"
#include <string.h>

#ifdef __cplusplus
	};
#endif

// NOLINTBEGIN(readability-*, bugprone-easily-swappable-parameters, clang-diagnostic-invalid-utf8, clang-diagnostic-invalid-source-encoding, clang-diagnostic-pointer-arith, clang-diagnostic-strict-prototypes, hicpp-uppercase-literal-suffix, cppcoreguidelines-*, performance-*)

/* Fügt eine Zeichenfolge in einen Text ein */
plcstring* BrbStringInsert(plcstring* pText, unsigned long nInsertIndex, plcstring* pInsert)
{
	STRING* pResult = 0;
	UDINT nTextLen = strlen(pText);
	UDINT nInsertLen = strlen(pInsert);
	UDINT nRestLen = nTextLen - nInsertIndex + 1;
	// Zeichen am Index nach hinten schieben
	memmove((pText + nInsertIndex + nInsertLen), (pText + nInsertIndex), nRestLen);
	memcpy((pText + nInsertIndex), pInsert, nInsertLen); // NOLINT(bugprone-not-null-terminated-result)
	pResult = pText + nInsertIndex + nInsertLen;
	return pResult;
}

// NOLINTEND(readability-*, bugprone-easily-swappable-parameters, clang-diagnostic-invalid-utf8, clang-diagnostic-invalid-source-encoding, clang-diagnostic-pointer-arith, clang-diagnostic-strict-prototypes, hicpp-uppercase-literal-suffix, cppcoreguidelines-*, performance-*)
```

#### BrbStringReplace.c - Ersetzt eine Zeichenfolge in einem Text durch eine andere
```c
/********************************************************************
 * COPYRIGHT -- Bernecker + Rainer
 ********************************************************************
 * Library: BrbLib
 * File: BrbStringReplace.c
 * Author: niedermeierr
 * Created: July 05, 2013
 ********************************************************************
 * Implementation of library BrbLib
 ********************************************************************/

#include <bur/plctypes.h>
#ifdef __cplusplus
	extern "C"
	{
#endif

#include "BrbLib.h"
#include <string.h>

#ifdef __cplusplus
	};
#endif

// NOLINTBEGIN(readability-*, bugprone-easily-swappable-parameters, clang-diagnostic-invalid-utf8, clang-diagnostic-invalid-source-encoding, clang-diagnostic-pointer-arith, clang-diagnostic-strict-prototypes, hicpp-uppercase-literal-suffix, cppcoreguidelines-*, performance-*)

/* Ersetzt eine Zeichenfolge in einem Text durch eine andere */
unsigned long BrbStringReplace(plcstring* pText, plcstring* pFind, plcstring* pReplace)
{
	UDINT nResult = 0;
	UDINT nTextLen = strlen(pText);
	UDINT nFindLen = strlen(pFind);
	UDINT nReplaceLen = strlen(pReplace);
	DINT nDiff = (DINT)nReplaceLen - (DINT)nFindLen;
	UDINT nCharIndex = 0;
	// Text von vorne nach hinten durchsuchen
	while(1==1)
	{
		// Textstelle vergleichen
		if(memcmp((pText + nCharIndex), pFind, nFindLen) == 0)
		{
			// Text gefunden
			if(nDiff > 0)
			{
				// Replace ist länger
				UDINT nRestLen = nTextLen - nCharIndex + 1;
				memmove((pText + nCharIndex + nDiff), (pText + nCharIndex), nRestLen);
				memcpy((pText + nCharIndex), pReplace, nReplaceLen);
				nTextLen += (UDINT)nDiff;
				nCharIndex += nReplaceLen;
				nResult += 1;
			}
			else if(nDiff < 0)
			{
				// Replace ist kürzer
				UDINT nRestLen = (UDINT)((DINT)nTextLen - (DINT)nCharIndex + nDiff + 1);
				memmove((pText + nCharIndex), (pText + nCharIndex - nDiff), nRestLen);
				memcpy((pText + nCharIndex), pReplace, nReplaceLen);
				nTextLen = (UDINT)((DINT)nTextLen + nDiff);
				nCharIndex += nReplaceLen;
				nResult += 1;
			}
			else
			{
				// Zeichenfolgen sind gleich lang
				memcpy((pText + nCharIndex), pReplace, nReplaceLen);
				nCharIndex += nReplaceLen;
				nResult += 1;
			}
		}
		else
		{
			nCharIndex += 1;
		}
		if(nCharIndex>=nTextLen)
		{
			break;
		}
	}
	return nResult;
}

// NOLINTEND(readability-*, bugprone-easily-swappable-parameters, clang-diagnostic-invalid-utf8, clang-diagnostic-invalid-source-encoding, clang-diagnostic-pointer-arith, clang-diagnostic-strict-prototypes, hicpp-uppercase-literal-suffix, cppcoreguidelines-*, performance-*)
```
